;FOLD ARCON WDAT1 LIN P3 Vel=0.5 m/s CPDAT1 Tool[1]:cmttorch Base[1]:vrashatel ;%{PE}
  ;FOLD Parameters ;%{h}
    ;Params IlfProvider=kukaroboter.arctech.arconlin; Kuka.IsGlobalPoint=False; Kuka.PointName=P3; Kuka.BlendingEnabled=False; Kuka.MoveDataName=CPDAT1; Kuka.VelocityPath=0.5; Kuka.CurrentCDSetIndex=0; Kuka.MovementParameterFieldEnabled=True; ArcTech.WdatVarName=WDAT1; ArcTech.Basic=3.4.3.1264
  ;ENDFOLD
  $BWDSTART = FALSE
  LDAT_ACT = LCPDAT1
  FDAT_ACT = FP3
  BAS(#CP_PARAMS, 0.5)
  SET_CD_PARAMS (0)
  TRIGGER WHEN DISTANCE = 1 DELAY = ArcGetDelay(#PreDefinition, WDAT1) DO ArcMainNG(#PreDefinition, WDAT1, WP3) PRIO = -1
  TRIGGER WHEN PATH = ArcGetPath(#OnTheFlyArcOn, WDAT1) DELAY = ArcGetDelay(#GasPreflow, WDAT1) DO ArcMainNG(#GasPreflow, WDAT1, WP3) PRIO = -1
  TRIGGER WHEN PATH = ArcGetPath(#OnTheFlyArcOn, WDAT1) DELAY = 0 DO ArcMainNG(#ArcOnMoveStd, WDAT1, WP3) PRIO = -1
  ArcMainNG(#ArcOnBeforeMoveStd, WDAT1, WP3)
  LIN XP3
  ArcMainNG(#ArcOnAfterMoveStd, WDAT1, WP3)
;ENDFOLD
   $VEL.CP = 0.060
   LIN  {X -8.829, Y -2.041, Z 0.700, A 0.000, B 0.000, C 0.000} C_DIS

;FOLD ARCOFF WDAT2 LIN P4 CPDAT2 Tool[1]:cmttorch Base[1]:vrashatel ;%{PE}
  ;FOLD Parameters ;%{h}
    ;Params IlfProvider=kukaroboter.arctech.arcofflin; Kuka.IsGlobalPoint=False; Kuka.PointName=P4; Kuka.BlendingEnabled=False; Kuka.MoveDataName=CPDAT2; Kuka.VelocityPath=0.01; Kuka.CurrentCDSetIndex=0; Kuka.MovementParameterFieldEnabled=True; ArcTech.WdatVarName=WDAT2; ArcTech.Basic=3.4.3.1264
  ;ENDFOLD
  $BWDSTART = FALSE
  LDAT_ACT = LCPDAT2
  FDAT_ACT = FP4
  BAS(#CP_PARAMS, gArcBasVelDefinition)
  SET_CD_PARAMS (0)
  TRIGGER WHEN PATH = ArcGetPath(#ArcOffBefore, WDAT2) DELAY = 0 DO ArcMainNG(#ArcOffBeforeOffStd, WDAT2, WP4) PRIO = -1
  TRIGGER WHEN PATH = ArcGetPath(#OnTheFlyArcOff, WDAT2) DELAY = 0 DO ArcMainNG(#ArcOffMoveStd, WDAT2, WP4) PRIO = -1
  ArcMainNG(#ArcOffBeforeMoveStd, WDAT2, WP4)
  LIN XP4
  ArcMainNG(#ArcOffAfterMoveStd, WDAT2, WP4)
;ENDFOLD
   $VEL.CP = 0.080
   LIN  {X -8.829, Y -2.607, Z 0.700, A 0.000, B 0.000, C 0.000} C_DIS

;FOLD ARCON WDAT1 LIN P3 Vel=0.5 m/s CPDAT1 Tool[1]:cmttorch Base[1]:vrashatel ;%{PE}
  ;FOLD Parameters ;%{h}
    ;Params IlfProvider=kukaroboter.arctech.arconlin; Kuka.IsGlobalPoint=False; Kuka.PointName=P3; Kuka.BlendingEnabled=False; Kuka.MoveDataName=CPDAT1; Kuka.VelocityPath=0.5; Kuka.CurrentCDSetIndex=0; Kuka.MovementParameterFieldEnabled=True; ArcTech.WdatVarName=WDAT1; ArcTech.Basic=3.4.3.1264
  ;ENDFOLD
  $BWDSTART = FALSE
  LDAT_ACT = LCPDAT1
  FDAT_ACT = FP3
  BAS(#CP_PARAMS, 0.5)
  SET_CD_PARAMS (0)
  TRIGGER WHEN DISTANCE = 1 DELAY = ArcGetDelay(#PreDefinition, WDAT1) DO ArcMainNG(#PreDefinition, WDAT1, WP3) PRIO = -1
  TRIGGER WHEN PATH = ArcGetPath(#OnTheFlyArcOn, WDAT1) DELAY = ArcGetDelay(#GasPreflow, WDAT1) DO ArcMainNG(#GasPreflow, WDAT1, WP3) PRIO = -1
  TRIGGER WHEN PATH = ArcGetPath(#OnTheFlyArcOn, WDAT1) DELAY = 0 DO ArcMainNG(#ArcOnMoveStd, WDAT1, WP3) PRIO = -1
  ArcMainNG(#ArcOnBeforeMoveStd, WDAT1, WP3)
  LIN XP3
  ArcMainNG(#ArcOnAfterMoveStd, WDAT1, WP3)
;ENDFOLD
   $VEL.CP = 0.060
   LIN  {X 2.607, Y 8.829, Z 0.700, A 0.000, B 0.000, C 0.000} C_DIS

;FOLD ARCOFF WDAT2 LIN P4 CPDAT2 Tool[1]:cmttorch Base[1]:vrashatel ;%{PE}
  ;FOLD Parameters ;%{h}
    ;Params IlfProvider=kukaroboter.arctech.arcofflin; Kuka.IsGlobalPoint=False; Kuka.PointName=P4; Kuka.BlendingEnabled=False; Kuka.MoveDataName=CPDAT2; Kuka.VelocityPath=0.01; Kuka.CurrentCDSetIndex=0; Kuka.MovementParameterFieldEnabled=True; ArcTech.WdatVarName=WDAT2; ArcTech.Basic=3.4.3.1264
  ;ENDFOLD
  $BWDSTART = FALSE
  LDAT_ACT = LCPDAT2
  FDAT_ACT = FP4
  BAS(#CP_PARAMS, gArcBasVelDefinition)
  SET_CD_PARAMS (0)
  TRIGGER WHEN PATH = ArcGetPath(#ArcOffBefore, WDAT2) DELAY = 0 DO ArcMainNG(#ArcOffBeforeOffStd, WDAT2, WP4) PRIO = -1
  TRIGGER WHEN PATH = ArcGetPath(#OnTheFlyArcOff, WDAT2) DELAY = 0 DO ArcMainNG(#ArcOffMoveStd, WDAT2, WP4) PRIO = -1
  ArcMainNG(#ArcOffBeforeMoveStd, WDAT2, WP4)
  LIN XP4
  ArcMainNG(#ArcOffAfterMoveStd, WDAT2, WP4)
;ENDFOLD
   $VEL.CP = 0.080
   LIN  {X 3.172, Y 8.829, Z 0.700, A 0.000, B 0.000, C 0.000} C_DIS

;FOLD ARCON WDAT1 LIN P3 Vel=0.5 m/s CPDAT1 Tool[1]:cmttorch Base[1]:vrashatel ;%{PE}
  ;FOLD Parameters ;%{h}
    ;Params IlfProvider=kukaroboter.arctech.arconlin; Kuka.IsGlobalPoint=False; Kuka.PointName=P3; Kuka.BlendingEnabled=False; Kuka.MoveDataName=CPDAT1; Kuka.VelocityPath=0.5; Kuka.CurrentCDSetIndex=0; Kuka.MovementParameterFieldEnabled=True; ArcTech.WdatVarName=WDAT1; ArcTech.Basic=3.4.3.1264
  ;ENDFOLD
  $BWDSTART = FALSE
  LDAT_ACT = LCPDAT1
  FDAT_ACT = FP3
  BAS(#CP_PARAMS, 0.5)
  SET_CD_PARAMS (0)
  TRIGGER WHEN DISTANCE = 1 DELAY = ArcGetDelay(#PreDefinition, WDAT1) DO ArcMainNG(#PreDefinition, WDAT1, WP3) PRIO = -1
  TRIGGER WHEN PATH = ArcGetPath(#OnTheFlyArcOn, WDAT1) DELAY = ArcGetDelay(#GasPreflow, WDAT1) DO ArcMainNG(#GasPreflow, WDAT1, WP3) PRIO = -1
  TRIGGER WHEN PATH = ArcGetPath(#OnTheFlyArcOn, WDAT1) DELAY = 0 DO ArcMainNG(#ArcOnMoveStd, WDAT1, WP3) PRIO = -1
  ArcMainNG(#ArcOnBeforeMoveStd, WDAT1, WP3)
  LIN XP3
  ArcMainNG(#ArcOnAfterMoveStd, WDAT1, WP3)
;ENDFOLD
   $VEL.CP = 0.060
   LIN  {X -8.829, Y -3.172, Z 0.700, A 0.000, B 0.000, C 0.000} C_DIS

;FOLD ARCOFF WDAT2 LIN P4 CPDAT2 Tool[1]:cmttorch Base[1]:vrashatel ;%{PE}
  ;FOLD Parameters ;%{h}
    ;Params IlfProvider=kukaroboter.arctech.arcofflin; Kuka.IsGlobalPoint=False; Kuka.PointName=P4; Kuka.BlendingEnabled=False; Kuka.MoveDataName=CPDAT2; Kuka.VelocityPath=0.01; Kuka.CurrentCDSetIndex=0; Kuka.MovementParameterFieldEnabled=True; ArcTech.WdatVarName=WDAT2; ArcTech.Basic=3.4.3.1264
  ;ENDFOLD
  $BWDSTART = FALSE
  LDAT_ACT = LCPDAT2
  FDAT_ACT = FP4
  BAS(#CP_PARAMS, gArcBasVelDefinition)
  SET_CD_PARAMS (0)
  TRIGGER WHEN PATH = ArcGetPath(#ArcOffBefore, WDAT2) DELAY = 0 DO ArcMainNG(#ArcOffBeforeOffStd, WDAT2, WP4) PRIO = -1
  TRIGGER WHEN PATH = ArcGetPath(#OnTheFlyArcOff, WDAT2) DELAY = 0 DO ArcMainNG(#ArcOffMoveStd, WDAT2, WP4) PRIO = -1
  ArcMainNG(#ArcOffBeforeMoveStd, WDAT2, WP4)
  LIN XP4
  ArcMainNG(#ArcOffAfterMoveStd, WDAT2, WP4)
;ENDFOLD
   $VEL.CP = 0.080
   LIN  {X -8.829, Y -3.738, Z 0.700, A 0.000, B 0.000, C 0.000} C_DIS

;FOLD ARCON WDAT1 LIN P3 Vel=0.5 m/s CPDAT1 Tool[1]:cmttorch Base[1]:vrashatel ;%{PE}
  ;FOLD Parameters ;%{h}
    ;Params IlfProvider=kukaroboter.arctech.arconlin; Kuka.IsGlobalPoint=False; Kuka.PointName=P3; Kuka.BlendingEnabled=False; Kuka.MoveDataName=CPDAT1; Kuka.VelocityPath=0.5; Kuka.CurrentCDSetIndex=0; Kuka.MovementParameterFieldEnabled=True; ArcTech.WdatVarName=WDAT1; ArcTech.Basic=3.4.3.1264
  ;ENDFOLD
  $BWDSTART = FALSE
  LDAT_ACT = LCPDAT1
  FDAT_ACT = FP3
  BAS(#CP_PARAMS, 0.5)
  SET_CD_PARAMS (0)
  TRIGGER WHEN DISTANCE = 1 DELAY = ArcGetDelay(#PreDefinition, WDAT1) DO ArcMainNG(#PreDefinition, WDAT1, WP3) PRIO = -1
  TRIGGER WHEN PATH = ArcGetPath(#OnTheFlyArcOn, WDAT1) DELAY = ArcGetDelay(#GasPreflow, WDAT1) DO ArcMainNG(#GasPreflow, WDAT1, WP3) PRIO = -1
  TRIGGER WHEN PATH = ArcGetPath(#OnTheFlyArcOn, WDAT1) DELAY = 0 DO ArcMainNG(#ArcOnMoveStd, WDAT1, WP3) PRIO = -1
  ArcMainNG(#ArcOnBeforeMoveStd, WDAT1, WP3)
  LIN XP3
  ArcMainNG(#ArcOnAfterMoveStd, WDAT1, WP3)
;ENDFOLD
   $VEL.CP = 0.060
   LIN  {X 3.738, Y 8.829, Z 0.700, A 0.000, B 0.000, C 0.000} C_DIS

;FOLD ARCOFF WDAT2 LIN P4 CPDAT2 Tool[1]:cmttorch Base[1]:vrashatel ;%{PE}
  ;FOLD Parameters ;%{h}
    ;Params IlfProvider=kukaroboter.arctech.arcofflin; Kuka.IsGlobalPoint=False; Kuka.PointName=P4; Kuka.BlendingEnabled=False; Kuka.MoveDataName=CPDAT2; Kuka.VelocityPath=0.01; Kuka.CurrentCDSetIndex=0; Kuka.MovementParameterFieldEnabled=True; ArcTech.WdatVarName=WDAT2; ArcTech.Basic=3.4.3.1264
  ;ENDFOLD
  $BWDSTART = FALSE
  LDAT_ACT = LCPDAT2
  FDAT_ACT = FP4
  BAS(#CP_PARAMS, gArcBasVelDefinition)
  SET_CD_PARAMS (0)
  TRIGGER WHEN PATH = ArcGetPath(#ArcOffBefore, WDAT2) DELAY = 0 DO ArcMainNG(#ArcOffBeforeOffStd, WDAT2, WP4) PRIO = -1
  TRIGGER WHEN PATH = ArcGetPath(#OnTheFlyArcOff, WDAT2) DELAY = 0 DO ArcMainNG(#ArcOffMoveStd, WDAT2, WP4) PRIO = -1
  ArcMainNG(#ArcOffBeforeMoveStd, WDAT2, WP4)
  LIN XP4
  ArcMainNG(#ArcOffAfterMoveStd, WDAT2, WP4)
;ENDFOLD
   $VEL.CP = 0.080
   LIN  {X 4.304, Y 8.829, Z 0.700, A 0.000, B 0.000, C 0.000} C_DIS

;FOLD ARCON WDAT1 LIN P3 Vel=0.5 m/s CPDAT1 Tool[1]:cmttorch Base[1]:vrashatel ;%{PE}
  ;FOLD Parameters ;%{h}
    ;Params IlfProvider=kukaroboter.arctech.arconlin; Kuka.IsGlobalPoint=False; Kuka.PointName=P3; Kuka.BlendingEnabled=False; Kuka.MoveDataName=CPDAT1; Kuka.VelocityPath=0.5; Kuka.CurrentCDSetIndex=0; Kuka.MovementParameterFieldEnabled=True; ArcTech.WdatVarName=WDAT1; ArcTech.Basic=3.4.3.1264
  ;ENDFOLD
  $BWDSTART = FALSE
  LDAT_ACT = LCPDAT1
  FDAT_ACT = FP3
  BAS(#CP_PARAMS, 0.5)
  SET_CD_PARAMS (0)
  TRIGGER WHEN DISTANCE = 1 DELAY = ArcGetDelay(#PreDefinition, WDAT1) DO ArcMainNG(#PreDefinition, WDAT1, WP3) PRIO = -1
  TRIGGER WHEN PATH = ArcGetPath(#OnTheFlyArcOn, WDAT1) DELAY = ArcGetDelay(#GasPreflow, WDAT1) DO ArcMainNG(#GasPreflow, WDAT1, WP3) PRIO = -1
  TRIGGER WHEN PATH = ArcGetPath(#OnTheFlyArcOn, WDAT1) DELAY = 0 DO ArcMainNG(#ArcOnMoveStd, WDAT1, WP3) PRIO = -1
  ArcMainNG(#ArcOnBeforeMoveStd, WDAT1, WP3)
  LIN XP3
  ArcMainNG(#ArcOnAfterMoveStd, WDAT1, WP3)
;ENDFOLD
   $VEL.CP = 0.060
   LIN  {X -8.829, Y -4.304, Z 0.700, A 0.000, B 0.000, C 0.000} C_DIS

;FOLD ARCOFF WDAT2 LIN P4 CPDAT2 Tool[1]:cmttorch Base[1]:vrashatel ;%{PE}
  ;FOLD Parameters ;%{h}
    ;Params IlfProvider=kukaroboter.arctech.arcofflin; Kuka.IsGlobalPoint=False; Kuka.PointName=P4; Kuka.BlendingEnabled=False; Kuka.MoveDataName=CPDAT2; Kuka.VelocityPath=0.01; Kuka.CurrentCDSetIndex=0; Kuka.MovementParameterFieldEnabled=True; ArcTech.WdatVarName=WDAT2; ArcTech.Basic=3.4.3.1264
  ;ENDFOLD
  $BWDSTART = FALSE
  LDAT_ACT = LCPDAT2
  FDAT_ACT = FP4
  BAS(#CP_PARAMS, gArcBasVelDefinition)
  SET_CD_PARAMS (0)
  TRIGGER WHEN PATH = ArcGetPath(#ArcOffBefore, WDAT2) DELAY = 0 DO ArcMainNG(#ArcOffBeforeOffStd, WDAT2, WP4) PRIO = -1
  TRIGGER WHEN PATH = ArcGetPath(#OnTheFlyArcOff, WDAT2) DELAY = 0 DO ArcMainNG(#ArcOffMoveStd, WDAT2, WP4) PRIO = -1
  ArcMainNG(#ArcOffBeforeMoveStd, WDAT2, WP4)
  LIN XP4
  ArcMainNG(#ArcOffAfterMoveStd, WDAT2, WP4)
;ENDFOLD
   $VEL.CP = 0.080
   LIN  {X -8.829, Y -4.869, Z 0.700, A 0.000, B 0.000, C 0.000} C_DIS

;FOLD ARCON WDAT1 LIN P3 Vel=0.5 m/s CPDAT1 Tool[1]:cmttorch Base[1]:vrashatel ;%{PE}
  ;FOLD Parameters ;%{h}
    ;Params IlfProvider=kukaroboter.arctech.arconlin; Kuka.IsGlobalPoint=False; Kuka.PointName=P3; Kuka.BlendingEnabled=False; Kuka.MoveDataName=CPDAT1; Kuka.VelocityPath=0.5; Kuka.CurrentCDSetIndex=0; Kuka.MovementParameterFieldEnabled=True; ArcTech.WdatVarName=WDAT1; ArcTech.Basic=3.4.3.1264
  ;ENDFOLD
  $BWDSTART = FALSE
  LDAT_ACT = LCPDAT1
  FDAT_ACT = FP3
  BAS(#CP_PARAMS, 0.5)
  SET_CD_PARAMS (0)
  TRIGGER WHEN DISTANCE = 1 DELAY = ArcGetDelay(#PreDefinition, WDAT1) DO ArcMainNG(#PreDefinition, WDAT1, WP3) PRIO = -1
  TRIGGER WHEN PATH = ArcGetPath(#OnTheFlyArcOn, WDAT1) DELAY = ArcGetDelay(#GasPreflow, WDAT1) DO ArcMainNG(#GasPreflow, WDAT1, WP3) PRIO = -1
  TRIGGER WHEN PATH = ArcGetPath(#OnTheFlyArcOn, WDAT1) DELAY = 0 DO ArcMainNG(#ArcOnMoveStd, WDAT1, WP3) PRIO = -1
  ArcMainNG(#ArcOnBeforeMoveStd, WDAT1, WP3)
  LIN XP3
  ArcMainNG(#ArcOnAfterMoveStd, WDAT1, WP3)
;ENDFOLD
   $VEL.CP = 0.060
   LIN  {X 4.869, Y 8.829, Z 0.700, A 0.000, B 0.000, C 0.000} C_DIS

;FOLD ARCOFF WDAT2 LIN P4 CPDAT2 Tool[1]:cmttorch Base[1]:vrashatel ;%{PE}
  ;FOLD Parameters ;%{h}
    ;Params IlfProvider=kukaroboter.arctech.arcofflin; Kuka.IsGlobalPoint=False; Kuka.PointName=P4; Kuka.BlendingEnabled=False; Kuka.MoveDataName=CPDAT2; Kuka.VelocityPath=0.01; Kuka.CurrentCDSetIndex=0; Kuka.MovementParameterFieldEnabled=True; ArcTech.WdatVarName=WDAT2; ArcTech.Basic=3.4.3.1264
  ;ENDFOLD
  $BWDSTART = FALSE
  LDAT_ACT = LCPDAT2
  FDAT_ACT = FP4
  BAS(#CP_PARAMS, gArcBasVelDefinition)
  SET_CD_PARAMS (0)
  TRIGGER WHEN PATH = ArcGetPath(#ArcOffBefore, WDAT2) DELAY = 0 DO ArcMainNG(#ArcOffBeforeOffStd, WDAT2, WP4) PRIO = -1
  TRIGGER WHEN PATH = ArcGetPath(#OnTheFlyArcOff, WDAT2) DELAY = 0 DO ArcMainNG(#ArcOffMoveStd, WDAT2, WP4) PRIO = -1
  ArcMainNG(#ArcOffBeforeMoveStd, WDAT2, WP4)
  LIN XP4
  ArcMainNG(#ArcOffAfterMoveStd, WDAT2, WP4)
;ENDFOLD
   $VEL.CP = 0.080
   LIN  {X 5.435, Y 8.829, Z 0.700, A 0.000, B 0.000, C 0.000} C_DIS

;FOLD ARCON WDAT1 LIN P3 Vel=0.5 m/s CPDAT1 Tool[1]:cmttorch Base[1]:vrashatel ;%{PE}
  ;FOLD Parameters ;%{h}
    ;Params IlfProvider=kukaroboter.arctech.arconlin; Kuka.IsGlobalPoint=False; Kuka.PointName=P3; Kuka.BlendingEnabled=False; Kuka.MoveDataName=CPDAT1; Kuka.VelocityPath=0.5; Kuka.CurrentCDSetIndex=0; Kuka.MovementParameterFieldEnabled=True; ArcTech.WdatVarName=WDAT1; ArcTech.Basic=3.4.3.1264
  ;ENDFOLD
  $BWDSTART = FALSE
  LDAT_ACT = LCPDAT1
  FDAT_ACT = FP3
  BAS(#CP_PARAMS, 0.5)
  SET_CD_PARAMS (0)
  TRIGGER WHEN DISTANCE = 1 DELAY = ArcGetDelay(#PreDefinition, WDAT1) DO ArcMainNG(#PreDefinition, WDAT1, WP3) PRIO = -1
  TRIGGER WHEN PATH = ArcGetPath(#OnTheFlyArcOn, WDAT1) DELAY = ArcGetDelay(#GasPreflow, WDAT1) DO ArcMainNG(#GasPreflow, WDAT1, WP3) PRIO = -1
  TRIGGER WHEN PATH = ArcGetPath(#OnTheFlyArcOn, WDAT1) DELAY = 0 DO ArcMainNG(#ArcOnMoveStd, WDAT1, WP3) PRIO = -1
  ArcMainNG(#ArcOnBeforeMoveStd, WDAT1, WP3)
  LIN XP3
  ArcMainNG(#ArcOnAfterMoveStd, WDAT1, WP3)
;ENDFOLD
   $VEL.CP = 0.060
   LIN  {X -8.829, Y -5.435, Z 0.700, A 0.000, B 0.000, C 0.000} C_DIS

;FOLD ARCOFF WDAT2 LIN P4 CPDAT2 Tool[1]:cmttorch Base[1]:vrashatel ;%{PE}
  ;FOLD Parameters ;%{h}
    ;Params IlfProvider=kukaroboter.arctech.arcofflin; Kuka.IsGlobalPoint=False; Kuka.PointName=P4; Kuka.BlendingEnabled=False; Kuka.MoveDataName=CPDAT2; Kuka.VelocityPath=0.01; Kuka.CurrentCDSetIndex=0; Kuka.MovementParameterFieldEnabled=True; ArcTech.WdatVarName=WDAT2; ArcTech.Basic=3.4.3.1264
  ;ENDFOLD
  $BWDSTART = FALSE
  LDAT_ACT = LCPDAT2
  FDAT_ACT = FP4
  BAS(#CP_PARAMS, gArcBasVelDefinition)
  SET_CD_PARAMS (0)
  TRIGGER WHEN PATH = ArcGetPath(#ArcOffBefore, WDAT2) DELAY = 0 DO ArcMainNG(#ArcOffBeforeOffStd, WDAT2, WP4) PRIO = -1
  TRIGGER WHEN PATH = ArcGetPath(#OnTheFlyArcOff, WDAT2) DELAY = 0 DO ArcMainNG(#ArcOffMoveStd, WDAT2, WP4) PRIO = -1
  ArcMainNG(#ArcOffBeforeMoveStd, WDAT2, WP4)
  LIN XP4
  ArcMainNG(#ArcOffAfterMoveStd, WDAT2, WP4)
;ENDFOLD
   $VEL.CP = 0.080
   LIN  {X -8.829, Y -6.001, Z 0.700, A 0.000, B 0.000, C 0.000} C_DIS

;FOLD ARCON WDAT1 LIN P3 Vel=0.5 m/s CPDAT1 Tool[1]:cmttorch Base[1]:vrashatel ;%{PE}
  ;FOLD Parameters ;%{h}
    ;Params IlfProvider=kukaroboter.arctech.arconlin; Kuka.IsGlobalPoint=False; Kuka.PointName=P3; Kuka.BlendingEnabled=False; Kuka.MoveDataName=CPDAT1; Kuka.VelocityPath=0.5; Kuka.CurrentCDSetIndex=0; Kuka.MovementParameterFieldEnabled=True; ArcTech.WdatVarName=WDAT1; ArcTech.Basic=3.4.3.1264
  ;ENDFOLD
  $BWDSTART = FALSE
  LDAT_ACT = LCPDAT1
  FDAT_ACT = FP3
  BAS(#CP_PARAMS, 0.5)
  SET_CD_PARAMS (0)
  TRIGGER WHEN DISTANCE = 1 DELAY = ArcGetDelay(#PreDefinition, WDAT1) DO ArcMainNG(#PreDefinition, WDAT1, WP3) PRIO = -1
  TRIGGER WHEN PATH = ArcGetPath(#OnTheFlyArcOn, WDAT1) DELAY = ArcGetDelay(#GasPreflow, WDAT1) DO ArcMainNG(#GasPreflow, WDAT1, WP3) PRIO = -1
  TRIGGER WHEN PATH = ArcGetPath(#OnTheFlyArcOn, WDAT1) DELAY = 0 DO ArcMainNG(#ArcOnMoveStd, WDAT1, WP3) PRIO = -1
  ArcMainNG(#ArcOnBeforeMoveStd, WDAT1, WP3)
  LIN XP3
  ArcMainNG(#ArcOnAfterMoveStd, WDAT1, WP3)
;ENDFOLD
   $VEL.CP = 0.060
   LIN  {X 6.001, Y 8.829, Z 0.700, A 0.000, B 0.000, C 0.000} C_DIS

;FOLD ARCOFF WDAT2 LIN P4 CPDAT2 Tool[1]:cmttorch Base[1]:vrashatel ;%{PE}
  ;FOLD Parameters ;%{h}
    ;Params IlfProvider=kukaroboter.arctech.arcofflin; Kuka.IsGlobalPoint=False; Kuka.PointName=P4; Kuka.BlendingEnabled=False; Kuka.MoveDataName=CPDAT2; Kuka.VelocityPath=0.01; Kuka.CurrentCDSetIndex=0; Kuka.MovementParameterFieldEnabled=True; ArcTech.WdatVarName=WDAT2; ArcTech.Basic=3.4.3.1264
  ;ENDFOLD
  $BWDSTART = FALSE
  LDAT_ACT = LCPDAT2
  FDAT_ACT = FP4
  BAS(#CP_PARAMS, gArcBasVelDefinition)
  SET_CD_PARAMS (0)
  TRIGGER WHEN PATH = ArcGetPath(#ArcOffBefore, WDAT2) DELAY = 0 DO ArcMainNG(#ArcOffBeforeOffStd, WDAT2, WP4) PRIO = -1
  TRIGGER WHEN PATH = ArcGetPath(#OnTheFlyArcOff, WDAT2) DELAY = 0 DO ArcMainNG(#ArcOffMoveStd, WDAT2, WP4) PRIO = -1
  ArcMainNG(#ArcOffBeforeMoveStd, WDAT2, WP4)
  LIN XP4
  ArcMainNG(#ArcOffAfterMoveStd, WDAT2, WP4)
;ENDFOLD
   $VEL.CP = 0.080
   LIN  {X 6.566, Y 8.829, Z 0.700, A 0.000, B 0.000, C 0.000} C_DIS

;FOLD ARCON WDAT1 LIN P3 Vel=0.5 m/s CPDAT1 Tool[1]:cmttorch Base[1]:vrashatel ;%{PE}
  ;FOLD Parameters ;%{h}
    ;Params IlfProvider=kukaroboter.arctech.arconlin; Kuka.IsGlobalPoint=False; Kuka.PointName=P3; Kuka.BlendingEnabled=False; Kuka.MoveDataName=CPDAT1; Kuka.VelocityPath=0.5; Kuka.CurrentCDSetIndex=0; Kuka.MovementParameterFieldEnabled=True; ArcTech.WdatVarName=WDAT1; ArcTech.Basic=3.4.3.1264
  ;ENDFOLD
  $BWDSTART = FALSE
  LDAT_ACT = LCPDAT1
  FDAT_ACT = FP3
  BAS(#CP_PARAMS, 0.5)
  SET_CD_PARAMS (0)
  TRIGGER WHEN DISTANCE = 1 DELAY = ArcGetDelay(#PreDefinition, WDAT1) DO ArcMainNG(#PreDefinition, WDAT1, WP3) PRIO = -1
  TRIGGER WHEN PATH = ArcGetPath(#OnTheFlyArcOn, WDAT1) DELAY = ArcGetDelay(#GasPreflow, WDAT1) DO ArcMainNG(#GasPreflow, WDAT1, WP3) PRIO = -1
  TRIGGER WHEN PATH = ArcGetPath(#OnTheFlyArcOn, WDAT1) DELAY = 0 DO ArcMainNG(#ArcOnMoveStd, WDAT1, WP3) PRIO = -1
  ArcMainNG(#ArcOnBeforeMoveStd, WDAT1, WP3)
  LIN XP3
  ArcMainNG(#ArcOnAfterMoveStd, WDAT1, WP3)
;ENDFOLD
   $VEL.CP = 0.060
   LIN  {X -8.829, Y -6.566, Z 0.700, A 0.000, B 0.000, C 0.000} C_DIS

;FOLD ARCOFF WDAT2 LIN P4 CPDAT2 Tool[1]:cmttorch Base[1]:vrashatel ;%{PE}
  ;FOLD Parameters ;%{h}
    ;Params IlfProvider=kukaroboter.arctech.arcofflin; Kuka.IsGlobalPoint=False; Kuka.PointName=P4; Kuka.BlendingEnabled=False; Kuka.MoveDataName=CPDAT2; Kuka.VelocityPath=0.01; Kuka.CurrentCDSetIndex=0; Kuka.MovementParameterFieldEnabled=True; ArcTech.WdatVarName=WDAT2; ArcTech.Basic=3.4.3.1264
  ;ENDFOLD
  $BWDSTART = FALSE
  LDAT_ACT = LCPDAT2
  FDAT_ACT = FP4
  BAS(#CP_PARAMS, gArcBasVelDefinition)
  SET_CD_PARAMS (0)
  TRIGGER WHEN PATH = ArcGetPath(#ArcOffBefore, WDAT2) DELAY = 0 DO ArcMainNG(#ArcOffBeforeOffStd, WDAT2, WP4) PRIO = -1
  TRIGGER WHEN PATH = ArcGetPath(#OnTheFlyArcOff, WDAT2) DELAY = 0 DO ArcMainNG(#ArcOffMoveStd, WDAT2, WP4) PRIO = -1
  ArcMainNG(#ArcOffBeforeMoveStd, WDAT2, WP4)
  LIN XP4
  ArcMainNG(#ArcOffAfterMoveStd, WDAT2, WP4)
;ENDFOLD
   $VEL.CP = 0.080
   LIN  {X -8.829, Y -7.132, Z 0.700, A 0.000, B 0.000, C 0.000} C_DIS

;FOLD ARCON WDAT1 LIN P3 Vel=0.5 m/s CPDAT1 Tool[1]:cmttorch Base[1]:vrashatel ;%{PE}
  ;FOLD Parameters ;%{h}
    ;Params IlfProvider=kukaroboter.arctech.arconlin; Kuka.IsGlobalPoint=False; Kuka.PointName=P3; Kuka.BlendingEnabled=False; Kuka.MoveDataName=CPDAT1; Kuka.VelocityPath=0.5; Kuka.CurrentCDSetIndex=0; Kuka.MovementParameterFieldEnabled=True; ArcTech.WdatVarName=WDAT1; ArcTech.Basic=3.4.3.1264
  ;ENDFOLD
  $BWDSTART = FALSE
  LDAT_ACT = LCPDAT1
  FDAT_ACT = FP3
  BAS(#CP_PARAMS, 0.5)
  SET_CD_PARAMS (0)
  TRIGGER WHEN DISTANCE = 1 DELAY = ArcGetDelay(#PreDefinition, WDAT1) DO ArcMainNG(#PreDefinition, WDAT1, WP3) PRIO = -1
  TRIGGER WHEN PATH = ArcGetPath(#OnTheFlyArcOn, WDAT1) DELAY = ArcGetDelay(#GasPreflow, WDAT1) DO ArcMainNG(#GasPreflow, WDAT1, WP3) PRIO = -1
  TRIGGER WHEN PATH = ArcGetPath(#OnTheFlyArcOn, WDAT1) DELAY = 0 DO ArcMainNG(#ArcOnMoveStd, WDAT1, WP3) PRIO = -1
  ArcMainNG(#ArcOnBeforeMoveStd, WDAT1, WP3)
  LIN XP3
  ArcMainNG(#ArcOnAfterMoveStd, WDAT1, WP3)
;ENDFOLD
   $VEL.CP = 0.060
   LIN  {X 7.132, Y 8.829, Z 0.700, A 0.000, B 0.000, C 0.000} C_DIS

;FOLD ARCOFF WDAT2 LIN P4 CPDAT2 Tool[1]:cmttorch Base[1]:vrashatel ;%{PE}
  ;FOLD Parameters ;%{h}
    ;Params IlfProvider=kukaroboter.arctech.arcofflin; Kuka.IsGlobalPoint=False; Kuka.PointName=P4; Kuka.BlendingEnabled=False; Kuka.MoveDataName=CPDAT2; Kuka.VelocityPath=0.01; Kuka.CurrentCDSetIndex=0; Kuka.MovementParameterFieldEnabled=True; ArcTech.WdatVarName=WDAT2; ArcTech.Basic=3.4.3.1264
  ;ENDFOLD
  $BWDSTART = FALSE
  LDAT_ACT = LCPDAT2
  FDAT_ACT = FP4
  BAS(#CP_PARAMS, gArcBasVelDefinition)
  SET_CD_PARAMS (0)
  TRIGGER WHEN PATH = ArcGetPath(#ArcOffBefore, WDAT2) DELAY = 0 DO ArcMainNG(#ArcOffBeforeOffStd, WDAT2, WP4) PRIO = -1
  TRIGGER WHEN PATH = ArcGetPath(#OnTheFlyArcOff, WDAT2) DELAY = 0 DO ArcMainNG(#ArcOffMoveStd, WDAT2, WP4) PRIO = -1
  ArcMainNG(#ArcOffBeforeMoveStd, WDAT2, WP4)
  LIN XP4
  ArcMainNG(#ArcOffAfterMoveStd, WDAT2, WP4)
;ENDFOLD
   $VEL.CP = 0.080
   LIN  {X 7.698, Y 8.829, Z 0.700, A 0.000, B 0.000, C 0.000} C_DIS

;FOLD ARCON WDAT1 LIN P3 Vel=0.5 m/s CPDAT1 Tool[1]:cmttorch Base[1]:vrashatel ;%{PE}
  ;FOLD Parameters ;%{h}
    ;Params IlfProvider=kukaroboter.arctech.arconlin; Kuka.IsGlobalPoint=False; Kuka.PointName=P3; Kuka.BlendingEnabled=False; Kuka.MoveDataName=CPDAT1; Kuka.VelocityPath=0.5; Kuka.CurrentCDSetIndex=0; Kuka.MovementParameterFieldEnabled=True; ArcTech.WdatVarName=WDAT1; ArcTech.Basic=3.4.3.1264
  ;ENDFOLD
  $BWDSTART = FALSE
  LDAT_ACT = LCPDAT1
  FDAT_ACT = FP3
  BAS(#CP_PARAMS, 0.5)
  SET_CD_PARAMS (0)
  TRIGGER WHEN DISTANCE = 1 DELAY = ArcGetDelay(#PreDefinition, WDAT1) DO ArcMainNG(#PreDefinition, WDAT1, WP3) PRIO = -1
  TRIGGER WHEN PATH = ArcGetPath(#OnTheFlyArcOn, WDAT1) DELAY = ArcGetDelay(#GasPreflow, WDAT1) DO ArcMainNG(#GasPreflow, WDAT1, WP3) PRIO = -1
  TRIGGER WHEN PATH = ArcGetPath(#OnTheFlyArcOn, WDAT1) DELAY = 0 DO ArcMainNG(#ArcOnMoveStd, WDAT1, WP3) PRIO = -1
  ArcMainNG(#ArcOnBeforeMoveStd, WDAT1, WP3)
  LIN XP3
  ArcMainNG(#ArcOnAfterMoveStd, WDAT1, WP3)
;ENDFOLD
   $VEL.CP = 0.060
   LIN  {X -8.829, Y -7.698, Z 0.700, A 0.000, B 0.000, C 0.000} C_DIS

;FOLD ARCOFF WDAT2 LIN P4 CPDAT2 Tool[1]:cmttorch Base[1]:vrashatel ;%{PE}
  ;FOLD Parameters ;%{h}
    ;Params IlfProvider=kukaroboter.arctech.arcofflin; Kuka.IsGlobalPoint=False; Kuka.PointName=P4; Kuka.BlendingEnabled=False; Kuka.MoveDataName=CPDAT2; Kuka.VelocityPath=0.01; Kuka.CurrentCDSetIndex=0; Kuka.MovementParameterFieldEnabled=True; ArcTech.WdatVarName=WDAT2; ArcTech.Basic=3.4.3.1264
  ;ENDFOLD
  $BWDSTART = FALSE
  LDAT_ACT = LCPDAT2
  FDAT_ACT = FP4
  BAS(#CP_PARAMS, gArcBasVelDefinition)
  SET_CD_PARAMS (0)
  TRIGGER WHEN PATH = ArcGetPath(#ArcOffBefore, WDAT2) DELAY = 0 DO ArcMainNG(#ArcOffBeforeOffStd, WDAT2, WP4) PRIO = -1
  TRIGGER WHEN PATH = ArcGetPath(#OnTheFlyArcOff, WDAT2) DELAY = 0 DO ArcMainNG(#ArcOffMoveStd, WDAT2, WP4) PRIO = -1
  ArcMainNG(#ArcOffBeforeMoveStd, WDAT2, WP4)
  LIN XP4
  ArcMainNG(#ArcOffAfterMoveStd, WDAT2, WP4)
;ENDFOLD
   $VEL.CP = 0.080
   LIN  {X -8.829, Y -8.263, Z 0.700, A 0.000, B 0.000, C 0.000} C_DIS

;FOLD ARCON WDAT1 LIN P3 Vel=0.5 m/s CPDAT1 Tool[1]:cmttorch Base[1]:vrashatel ;%{PE}
  ;FOLD Parameters ;%{h}
    ;Params IlfProvider=kukaroboter.arctech.arconlin; Kuka.IsGlobalPoint=False; Kuka.PointName=P3; Kuka.BlendingEnabled=False; Kuka.MoveDataName=CPDAT1; Kuka.VelocityPath=0.5; Kuka.CurrentCDSetIndex=0; Kuka.MovementParameterFieldEnabled=True; ArcTech.WdatVarName=WDAT1; ArcTech.Basic=3.4.3.1264
  ;ENDFOLD
  $BWDSTART = FALSE
  LDAT_ACT = LCPDAT1
  FDAT_ACT = FP3
  BAS(#CP_PARAMS, 0.5)
  SET_CD_PARAMS (0)
  TRIGGER WHEN DISTANCE = 1 DELAY = ArcGetDelay(#PreDefinition, WDAT1) DO ArcMainNG(#PreDefinition, WDAT1, WP3) PRIO = -1
  TRIGGER WHEN PATH = ArcGetPath(#OnTheFlyArcOn, WDAT1) DELAY = ArcGetDelay(#GasPreflow, WDAT1) DO ArcMainNG(#GasPreflow, WDAT1, WP3) PRIO = -1
  TRIGGER WHEN PATH = ArcGetPath(#OnTheFlyArcOn, WDAT1) DELAY = 0 DO ArcMainNG(#ArcOnMoveStd, WDAT1, WP3) PRIO = -1
  ArcMainNG(#ArcOnBeforeMoveStd, WDAT1, WP3)
  LIN XP3
  ArcMainNG(#ArcOnAfterMoveStd, WDAT1, WP3)
;ENDFOLD
   $VEL.CP = 0.060
   LIN  {X 8.263, Y 8.829, Z 0.700, A 0.000, B 0.000, C 0.000} C_DIS

;FOLD ARCOFF WDAT2 LIN P4 CPDAT2 Tool[1]:cmttorch Base[1]:vrashatel ;%{PE}
  ;FOLD Parameters ;%{h}
    ;Params IlfProvider=kukaroboter.arctech.arcofflin; Kuka.IsGlobalPoint=False; Kuka.PointName=P4; Kuka.BlendingEnabled=False; Kuka.MoveDataName=CPDAT2; Kuka.VelocityPath=0.01; Kuka.CurrentCDSetIndex=0; Kuka.MovementParameterFieldEnabled=True; ArcTech.WdatVarName=WDAT2; ArcTech.Basic=3.4.3.1264
  ;ENDFOLD
  $BWDSTART = FALSE
  LDAT_ACT = LCPDAT2
  FDAT_ACT = FP4
  BAS(#CP_PARAMS, gArcBasVelDefinition)
  SET_CD_PARAMS (0)
  TRIGGER WHEN PATH = ArcGetPath(#ArcOffBefore, WDAT2) DELAY = 0 DO ArcMainNG(#ArcOffBeforeOffStd, WDAT2, WP4) PRIO = -1
  TRIGGER WHEN PATH = ArcGetPath(#OnTheFlyArcOff, WDAT2) DELAY = 0 DO ArcMainNG(#ArcOffMoveStd, WDAT2, WP4) PRIO = -1
  ArcMainNG(#ArcOffBeforeMoveStd, WDAT2, WP4)
  LIN XP4
  ArcMainNG(#ArcOffAfterMoveStd, WDAT2, WP4)
;ENDFOLD
   $VEL.CP = 0.080
   LIN  {X 8.829, Y 8.829, Z 0.700, A 0.000, B 0.000, C 0.000} C_DIS

;FOLD ARCON WDAT1 LIN P3 Vel=0.5 m/s CPDAT1 Tool[1]:cmttorch Base[1]:vrashatel ;%{PE}
  ;FOLD Parameters ;%{h}
    ;Params IlfProvider=kukaroboter.arctech.arconlin; Kuka.IsGlobalPoint=False; Kuka.PointName=P3; Kuka.BlendingEnabled=False; Kuka.MoveDataName=CPDAT1; Kuka.VelocityPath=0.5; Kuka.CurrentCDSetIndex=0; Kuka.MovementParameterFieldEnabled=True; ArcTech.WdatVarName=WDAT1; ArcTech.Basic=3.4.3.1264
  ;ENDFOLD
  $BWDSTART = FALSE
  LDAT_ACT = LCPDAT1
  FDAT_ACT = FP3
  BAS(#CP_PARAMS, 0.5)
  SET_CD_PARAMS (0)
  TRIGGER WHEN DISTANCE = 1 DELAY = ArcGetDelay(#PreDefinition, WDAT1) DO ArcMainNG(#PreDefinition, WDAT1, WP3) PRIO = -1
  TRIGGER WHEN PATH = ArcGetPath(#OnTheFlyArcOn, WDAT1) DELAY = ArcGetDelay(#GasPreflow, WDAT1) DO ArcMainNG(#GasPreflow, WDAT1, WP3) PRIO = -1
  TRIGGER WHEN PATH = ArcGetPath(#OnTheFlyArcOn, WDAT1) DELAY = 0 DO ArcMainNG(#ArcOnMoveStd, WDAT1, WP3) PRIO = -1
  ArcMainNG(#ArcOnBeforeMoveStd, WDAT1, WP3)
  LIN XP3
  ArcMainNG(#ArcOnAfterMoveStd, WDAT1, WP3)
;ENDFOLD
   $VEL.CP = 0.060
   LIN  {X -8.829, Y -8.829, Z 0.700, A 0.000, B 0.000, C 0.000} C_DIS

;FOLD ARCOFF WDAT2 LIN P4 CPDAT2 Tool[1]:cmttorch Base[1]:vrashatel ;%{PE}
  ;FOLD Parameters ;%{h}
    ;Params IlfProvider=kukaroboter.arctech.arcofflin; Kuka.IsGlobalPoint=False; Kuka.PointName=P4; Kuka.BlendingEnabled=False; Kuka.MoveDataName=CPDAT2; Kuka.VelocityPath=0.01; Kuka.CurrentCDSetIndex=0; Kuka.MovementParameterFieldEnabled=True; ArcTech.WdatVarName=WDAT2; ArcTech.Basic=3.4.3.1264
  ;ENDFOLD
  $BWDSTART = FALSE
  LDAT_ACT = LCPDAT2
  FDAT_ACT = FP4
  BAS(#CP_PARAMS, gArcBasVelDefinition)
  SET_CD_PARAMS (0)
  TRIGGER WHEN PATH = ArcGetPath(#ArcOffBefore, WDAT2) DELAY = 0 DO ArcMainNG(#ArcOffBeforeOffStd, WDAT2, WP4) PRIO = -1
  TRIGGER WHEN PATH = ArcGetPath(#OnTheFlyArcOff, WDAT2) DELAY = 0 DO ArcMainNG(#ArcOffMoveStd, WDAT2, WP4) PRIO = -1
  ArcMainNG(#ArcOffBeforeMoveStd, WDAT2, WP4)
  LIN XP4
  ArcMainNG(#ArcOffAfterMoveStd, WDAT2, WP4)
;ENDFOLD
   $VEL.CP = 0.080
   LIN  {X -8.263, Y -8.829, Z 0.700, A 0.000, B 0.000, C 0.000} C_DIS

;FOLD ARCON WDAT1 LIN P3 Vel=0.5 m/s CPDAT1 Tool[1]:cmttorch Base[1]:vrashatel ;%{PE}
  ;FOLD Parameters ;%{h}
    ;Params IlfProvider=kukaroboter.arctech.arconlin; Kuka.IsGlobalPoint=False; Kuka.PointName=P3; Kuka.BlendingEnabled=False; Kuka.MoveDataName=CPDAT1; Kuka.VelocityPath=0.5; Kuka.CurrentCDSetIndex=0; Kuka.MovementParameterFieldEnabled=True; ArcTech.WdatVarName=WDAT1; ArcTech.Basic=3.4.3.1264
  ;ENDFOLD
  $BWDSTART = FALSE
  LDAT_ACT = LCPDAT1
  FDAT_ACT = FP3
  BAS(#CP_PARAMS, 0.5)
  SET_CD_PARAMS (0)
  TRIGGER WHEN DISTANCE = 1 DELAY = ArcGetDelay(#PreDefinition, WDAT1) DO ArcMainNG(#PreDefinition, WDAT1, WP3) PRIO = -1
  TRIGGER WHEN PATH = ArcGetPath(#OnTheFlyArcOn, WDAT1) DELAY = ArcGetDelay(#GasPreflow, WDAT1) DO ArcMainNG(#GasPreflow, WDAT1, WP3) PRIO = -1
  TRIGGER WHEN PATH = ArcGetPath(#OnTheFlyArcOn, WDAT1) DELAY = 0 DO ArcMainNG(#ArcOnMoveStd, WDAT1, WP3) PRIO = -1
  ArcMainNG(#ArcOnBeforeMoveStd, WDAT1, WP3)
  LIN XP3
  ArcMainNG(#ArcOnAfterMoveStd, WDAT1, WP3)
;ENDFOLD
   $VEL.CP = 0.060
   LIN  {X 8.829, Y 8.263, Z 0.700, A 0.000, B 0.000, C 0.000} C_DIS

;FOLD ARCOFF WDAT2 LIN P4 CPDAT2 Tool[1]:cmttorch Base[1]:vrashatel ;%{PE}
  ;FOLD Parameters ;%{h}
    ;Params IlfProvider=kukaroboter.arctech.arcofflin; Kuka.IsGlobalPoint=False; Kuka.PointName=P4; Kuka.BlendingEnabled=False; Kuka.MoveDataName=CPDAT2; Kuka.VelocityPath=0.01; Kuka.CurrentCDSetIndex=0; Kuka.MovementParameterFieldEnabled=True; ArcTech.WdatVarName=WDAT2; ArcTech.Basic=3.4.3.1264
  ;ENDFOLD
  $BWDSTART = FALSE
  LDAT_ACT = LCPDAT2
  FDAT_ACT = FP4
  BAS(#CP_PARAMS, gArcBasVelDefinition)
  SET_CD_PARAMS (0)
  TRIGGER WHEN PATH = ArcGetPath(#ArcOffBefore, WDAT2) DELAY = 0 DO ArcMainNG(#ArcOffBeforeOffStd, WDAT2, WP4) PRIO = -1
  TRIGGER WHEN PATH = ArcGetPath(#OnTheFlyArcOff, WDAT2) DELAY = 0 DO ArcMainNG(#ArcOffMoveStd, WDAT2, WP4) PRIO = -1
  ArcMainNG(#ArcOffBeforeMoveStd, WDAT2, WP4)
  LIN XP4
  ArcMainNG(#ArcOffAfterMoveStd, WDAT2, WP4)
;ENDFOLD
   $VEL.CP = 0.080
   LIN  {X 8.829, Y 7.698, Z 0.700, A 0.000, B 0.000, C 0.000} C_DIS

;FOLD ARCON WDAT1 LIN P3 Vel=0.5 m/s CPDAT1 Tool[1]:cmttorch Base[1]:vrashatel ;%{PE}
  ;FOLD Parameters ;%{h}
    ;Params IlfProvider=kukaroboter.arctech.arconlin; Kuka.IsGlobalPoint=False; Kuka.PointName=P3; Kuka.BlendingEnabled=False; Kuka.MoveDataName=CPDAT1; Kuka.VelocityPath=0.5; Kuka.CurrentCDSetIndex=0; Kuka.MovementParameterFieldEnabled=True; ArcTech.WdatVarName=WDAT1; ArcTech.Basic=3.4.3.1264
  ;ENDFOLD
  $BWDSTART = FALSE
  LDAT_ACT = LCPDAT1
  FDAT_ACT = FP3
  BAS(#CP_PARAMS, 0.5)
  SET_CD_PARAMS (0)
  TRIGGER WHEN DISTANCE = 1 DELAY = ArcGetDelay(#PreDefinition, WDAT1) DO ArcMainNG(#PreDefinition, WDAT1, WP3) PRIO = -1
  TRIGGER WHEN PATH = ArcGetPath(#OnTheFlyArcOn, WDAT1) DELAY = ArcGetDelay(#GasPreflow, WDAT1) DO ArcMainNG(#GasPreflow, WDAT1, WP3) PRIO = -1
  TRIGGER WHEN PATH = ArcGetPath(#OnTheFlyArcOn, WDAT1) DELAY = 0 DO ArcMainNG(#ArcOnMoveStd, WDAT1, WP3) PRIO = -1
  ArcMainNG(#ArcOnBeforeMoveStd, WDAT1, WP3)
  LIN XP3
  ArcMainNG(#ArcOnAfterMoveStd, WDAT1, WP3)
;ENDFOLD
   $VEL.CP = 0.060
   LIN  {X -7.698, Y -8.829, Z 0.700, A 0.000, B 0.000, C 0.000} C_DIS

;FOLD ARCOFF WDAT2 LIN P4 CPDAT2 Tool[1]:cmttorch Base[1]:vrashatel ;%{PE}
  ;FOLD Parameters ;%{h}
    ;Params IlfProvider=kukaroboter.arctech.arcofflin; Kuka.IsGlobalPoint=False; Kuka.PointName=P4; Kuka.BlendingEnabled=False; Kuka.MoveDataName=CPDAT2; Kuka.VelocityPath=0.01; Kuka.CurrentCDSetIndex=0; Kuka.MovementParameterFieldEnabled=True; ArcTech.WdatVarName=WDAT2; ArcTech.Basic=3.4.3.1264
  ;ENDFOLD
  $BWDSTART = FALSE
  LDAT_ACT = LCPDAT2
  FDAT_ACT = FP4
  BAS(#CP_PARAMS, gArcBasVelDefinition)
  SET_CD_PARAMS (0)
  TRIGGER WHEN PATH = ArcGetPath(#ArcOffBefore, WDAT2) DELAY = 0 DO ArcMainNG(#ArcOffBeforeOffStd, WDAT2, WP4) PRIO = -1
  TRIGGER WHEN PATH = ArcGetPath(#OnTheFlyArcOff, WDAT2) DELAY = 0 DO ArcMainNG(#ArcOffMoveStd, WDAT2, WP4) PRIO = -1
  ArcMainNG(#ArcOffBeforeMoveStd, WDAT2, WP4)
  LIN XP4
  ArcMainNG(#ArcOffAfterMoveStd, WDAT2, WP4)
;ENDFOLD
   $VEL.CP = 0.080
   LIN  {X -7.132, Y -8.829, Z 0.700, A 0.000, B 0.000, C 0.000} C_DIS

;FOLD ARCON WDAT1 LIN P3 Vel=0.5 m/s CPDAT1 Tool[1]:cmttorch Base[1]:vrashatel ;%{PE}
  ;FOLD Parameters ;%{h}
    ;Params IlfProvider=kukaroboter.arctech.arconlin; Kuka.IsGlobalPoint=False; Kuka.PointName=P3; Kuka.BlendingEnabled=False; Kuka.MoveDataName=CPDAT1; Kuka.VelocityPath=0.5; Kuka.CurrentCDSetIndex=0; Kuka.MovementParameterFieldEnabled=True; ArcTech.WdatVarName=WDAT1; ArcTech.Basic=3.4.3.1264
  ;ENDFOLD
  $BWDSTART = FALSE
  LDAT_ACT = LCPDAT1
  FDAT_ACT = FP3
  BAS(#CP_PARAMS, 0.5)
  SET_CD_PARAMS (0)
  TRIGGER WHEN DISTANCE = 1 DELAY = ArcGetDelay(#PreDefinition, WDAT1) DO ArcMainNG(#PreDefinition, WDAT1, WP3) PRIO = -1
  TRIGGER WHEN PATH = ArcGetPath(#OnTheFlyArcOn, WDAT1) DELAY = ArcGetDelay(#GasPreflow, WDAT1) DO ArcMainNG(#GasPreflow, WDAT1, WP3) PRIO = -1
  TRIGGER WHEN PATH = ArcGetPath(#OnTheFlyArcOn, WDAT1) DELAY = 0 DO ArcMainNG(#ArcOnMoveStd, WDAT1, WP3) PRIO = -1
  ArcMainNG(#ArcOnBeforeMoveStd, WDAT1, WP3)
  LIN XP3
  ArcMainNG(#ArcOnAfterMoveStd, WDAT1, WP3)
;ENDFOLD
   $VEL.CP = 0.060
   LIN  {X 8.829, Y 7.132, Z 0.700, A 0.000, B 0.000, C 0.000} C_DIS

;FOLD ARCOFF WDAT2 LIN P4 CPDAT2 Tool[1]:cmttorch Base[1]:vrashatel ;%{PE}
  ;FOLD Parameters ;%{h}
    ;Params IlfProvider=kukaroboter.arctech.arcofflin; Kuka.IsGlobalPoint=False; Kuka.PointName=P4; Kuka.BlendingEnabled=False; Kuka.MoveDataName=CPDAT2; Kuka.VelocityPath=0.01; Kuka.CurrentCDSetIndex=0; Kuka.MovementParameterFieldEnabled=True; ArcTech.WdatVarName=WDAT2; ArcTech.Basic=3.4.3.1264
  ;ENDFOLD
  $BWDSTART = FALSE
  LDAT_ACT = LCPDAT2
  FDAT_ACT = FP4
  BAS(#CP_PARAMS, gArcBasVelDefinition)
  SET_CD_PARAMS (0)
  TRIGGER WHEN PATH = ArcGetPath(#ArcOffBefore, WDAT2) DELAY = 0 DO ArcMainNG(#ArcOffBeforeOffStd, WDAT2, WP4) PRIO = -1
  TRIGGER WHEN PATH = ArcGetPath(#OnTheFlyArcOff, WDAT2) DELAY = 0 DO ArcMainNG(#ArcOffMoveStd, WDAT2, WP4) PRIO = -1
  ArcMainNG(#ArcOffBeforeMoveStd, WDAT2, WP4)
  LIN XP4
  ArcMainNG(#ArcOffAfterMoveStd, WDAT2, WP4)
;ENDFOLD
   $VEL.CP = 0.080
   LIN  {X 8.829, Y 6.566, Z 0.700, A 0.000, B 0.000, C 0.000} C_DIS

;FOLD ARCON WDAT1 LIN P3 Vel=0.5 m/s CPDAT1 Tool[1]:cmttorch Base[1]:vrashatel ;%{PE}
  ;FOLD Parameters ;%{h}
    ;Params IlfProvider=kukaroboter.arctech.arconlin; Kuka.IsGlobalPoint=False; Kuka.PointName=P3; Kuka.BlendingEnabled=False; Kuka.MoveDataName=CPDAT1; Kuka.VelocityPath=0.5; Kuka.CurrentCDSetIndex=0; Kuka.MovementParameterFieldEnabled=True; ArcTech.WdatVarName=WDAT1; ArcTech.Basic=3.4.3.1264
  ;ENDFOLD
  $BWDSTART = FALSE
  LDAT_ACT = LCPDAT1
  FDAT_ACT = FP3
  BAS(#CP_PARAMS, 0.5)
  SET_CD_PARAMS (0)
  TRIGGER WHEN DISTANCE = 1 DELAY = ArcGetDelay(#PreDefinition, WDAT1) DO ArcMainNG(#PreDefinition, WDAT1, WP3) PRIO = -1
  TRIGGER WHEN PATH = ArcGetPath(#OnTheFlyArcOn, WDAT1) DELAY = ArcGetDelay(#GasPreflow, WDAT1) DO ArcMainNG(#GasPreflow, WDAT1, WP3) PRIO = -1
  TRIGGER WHEN PATH = ArcGetPath(#OnTheFlyArcOn, WDAT1) DELAY = 0 DO ArcMainNG(#ArcOnMoveStd, WDAT1, WP3) PRIO = -1
  ArcMainNG(#ArcOnBeforeMoveStd, WDAT1, WP3)
  LIN XP3
  ArcMainNG(#ArcOnAfterMoveStd, WDAT1, WP3)
;ENDFOLD
   $VEL.CP = 0.060
   LIN  {X -6.566, Y -8.829, Z 0.700, A 0.000, B 0.000, C 0.000} C_DIS

;FOLD ARCOFF WDAT2 LIN P4 CPDAT2 Tool[1]:cmttorch Base[1]:vrashatel ;%{PE}
  ;FOLD Parameters ;%{h}
    ;Params IlfProvider=kukaroboter.arctech.arcofflin; Kuka.IsGlobalPoint=False; Kuka.PointName=P4; Kuka.BlendingEnabled=False; Kuka.MoveDataName=CPDAT2; Kuka.VelocityPath=0.01; Kuka.CurrentCDSetIndex=0; Kuka.MovementParameterFieldEnabled=True; ArcTech.WdatVarName=WDAT2; ArcTech.Basic=3.4.3.1264
  ;ENDFOLD
  $BWDSTART = FALSE
  LDAT_ACT = LCPDAT2
  FDAT_ACT = FP4
  BAS(#CP_PARAMS, gArcBasVelDefinition)
  SET_CD_PARAMS (0)
  TRIGGER WHEN PATH = ArcGetPath(#ArcOffBefore, WDAT2) DELAY = 0 DO ArcMainNG(#ArcOffBeforeOffStd, WDAT2, WP4) PRIO = -1
  TRIGGER WHEN PATH = ArcGetPath(#OnTheFlyArcOff, WDAT2) DELAY = 0 DO ArcMainNG(#ArcOffMoveStd, WDAT2, WP4) PRIO = -1
  ArcMainNG(#ArcOffBeforeMoveStd, WDAT2, WP4)
  LIN XP4
  ArcMainNG(#ArcOffAfterMoveStd, WDAT2, WP4)
;ENDFOLD
   $VEL.CP = 0.080
   LIN  {X -6.001, Y -8.829, Z 0.700, A 0.000, B 0.000, C 0.000} C_DIS

;FOLD ARCON WDAT1 LIN P3 Vel=0.5 m/s CPDAT1 Tool[1]:cmttorch Base[1]:vrashatel ;%{PE}
  ;FOLD Parameters ;%{h}
    ;Params IlfProvider=kukaroboter.arctech.arconlin; Kuka.IsGlobalPoint=False; Kuka.PointName=P3; Kuka.BlendingEnabled=False; Kuka.MoveDataName=CPDAT1; Kuka.VelocityPath=0.5; Kuka.CurrentCDSetIndex=0; Kuka.MovementParameterFieldEnabled=True; ArcTech.WdatVarName=WDAT1; ArcTech.Basic=3.4.3.1264
  ;ENDFOLD
  $BWDSTART = FALSE
  LDAT_ACT = LCPDAT1
  FDAT_ACT = FP3
  BAS(#CP_PARAMS, 0.5)
  SET_CD_PARAMS (0)
  TRIGGER WHEN DISTANCE = 1 DELAY = ArcGetDelay(#PreDefinition, WDAT1) DO ArcMainNG(#PreDefinition, WDAT1, WP3) PRIO = -1
  TRIGGER WHEN PATH = ArcGetPath(#OnTheFlyArcOn, WDAT1) DELAY = ArcGetDelay(#GasPreflow, WDAT1) DO ArcMainNG(#GasPreflow, WDAT1, WP3) PRIO = -1
  TRIGGER WHEN PATH = ArcGetPath(#OnTheFlyArcOn, WDAT1) DELAY = 0 DO ArcMainNG(#ArcOnMoveStd, WDAT1, WP3) PRIO = -1
  ArcMainNG(#ArcOnBeforeMoveStd, WDAT1, WP3)
  LIN XP3
  ArcMainNG(#ArcOnAfterMoveStd, WDAT1, WP3)
;ENDFOLD
   $VEL.CP = 0.060
   LIN  {X 8.829, Y 6.001, Z 0.700, A 0.000, B 0.000, C 0.000} C_DIS

;FOLD ARCOFF WDAT2 LIN P4 CPDAT2 Tool[1]:cmttorch Base[1]:vrashatel ;%{PE}
  ;FOLD Parameters ;%{h}
    ;Params IlfProvider=kukaroboter.arctech.arcofflin; Kuka.IsGlobalPoint=False; Kuka.PointName=P4; Kuka.BlendingEnabled=False; Kuka.MoveDataName=CPDAT2; Kuka.VelocityPath=0.01; Kuka.CurrentCDSetIndex=0; Kuka.MovementParameterFieldEnabled=True; ArcTech.WdatVarName=WDAT2; ArcTech.Basic=3.4.3.1264
  ;ENDFOLD
  $BWDSTART = FALSE
  LDAT_ACT = LCPDAT2
  FDAT_ACT = FP4
  BAS(#CP_PARAMS, gArcBasVelDefinition)
  SET_CD_PARAMS (0)
  TRIGGER WHEN PATH = ArcGetPath(#ArcOffBefore, WDAT2) DELAY = 0 DO ArcMainNG(#ArcOffBeforeOffStd, WDAT2, WP4) PRIO = -1
  TRIGGER WHEN PATH = ArcGetPath(#OnTheFlyArcOff, WDAT2) DELAY = 0 DO ArcMainNG(#ArcOffMoveStd, WDAT2, WP4) PRIO = -1
  ArcMainNG(#ArcOffBeforeMoveStd, WDAT2, WP4)
  LIN XP4
  ArcMainNG(#ArcOffAfterMoveStd, WDAT2, WP4)
;ENDFOLD
   $VEL.CP = 0.080
   LIN  {X 8.829, Y 5.435, Z 0.700, A 0.000, B 0.000, C 0.000} C_DIS

;FOLD ARCON WDAT1 LIN P3 Vel=0.5 m/s CPDAT1 Tool[1]:cmttorch Base[1]:vrashatel ;%{PE}
  ;FOLD Parameters ;%{h}
    ;Params IlfProvider=kukaroboter.arctech.arconlin; Kuka.IsGlobalPoint=False; Kuka.PointName=P3; Kuka.BlendingEnabled=False; Kuka.MoveDataName=CPDAT1; Kuka.VelocityPath=0.5; Kuka.CurrentCDSetIndex=0; Kuka.MovementParameterFieldEnabled=True; ArcTech.WdatVarName=WDAT1; ArcTech.Basic=3.4.3.1264
  ;ENDFOLD
  $BWDSTART = FALSE
  LDAT_ACT = LCPDAT1
  FDAT_ACT = FP3
  BAS(#CP_PARAMS, 0.5)
  SET_CD_PARAMS (0)
  TRIGGER WHEN DISTANCE = 1 DELAY = ArcGetDelay(#PreDefinition, WDAT1) DO ArcMainNG(#PreDefinition, WDAT1, WP3) PRIO = -1
  TRIGGER WHEN PATH = ArcGetPath(#OnTheFlyArcOn, WDAT1) DELAY = ArcGetDelay(#GasPreflow, WDAT1) DO ArcMainNG(#GasPreflow, WDAT1, WP3) PRIO = -1
  TRIGGER WHEN PATH = ArcGetPath(#OnTheFlyArcOn, WDAT1) DELAY = 0 DO ArcMainNG(#ArcOnMoveStd, WDAT1, WP3) PRIO = -1
  ArcMainNG(#ArcOnBeforeMoveStd, WDAT1, WP3)
  LIN XP3
  ArcMainNG(#ArcOnAfterMoveStd, WDAT1, WP3)
;ENDFOLD
   $VEL.CP = 0.060
   LIN  {X -5.435, Y -8.829, Z 0.700, A 0.000, B 0.000, C 0.000} C_DIS

;FOLD ARCOFF WDAT2 LIN P4 CPDAT2 Tool[1]:cmttorch Base[1]:vrashatel ;%{PE}
  ;FOLD Parameters ;%{h}
    ;Params IlfProvider=kukaroboter.arctech.arcofflin; Kuka.IsGlobalPoint=False; Kuka.PointName=P4; Kuka.BlendingEnabled=False; Kuka.MoveDataName=CPDAT2; Kuka.VelocityPath=0.01; Kuka.CurrentCDSetIndex=0; Kuka.MovementParameterFieldEnabled=True; ArcTech.WdatVarName=WDAT2; ArcTech.Basic=3.4.3.1264
  ;ENDFOLD
  $BWDSTART = FALSE
  LDAT_ACT = LCPDAT2
  FDAT_ACT = FP4
  BAS(#CP_PARAMS, gArcBasVelDefinition)
  SET_CD_PARAMS (0)
  TRIGGER WHEN PATH = ArcGetPath(#ArcOffBefore, WDAT2) DELAY = 0 DO ArcMainNG(#ArcOffBeforeOffStd, WDAT2, WP4) PRIO = -1
  TRIGGER WHEN PATH = ArcGetPath(#OnTheFlyArcOff, WDAT2) DELAY = 0 DO ArcMainNG(#ArcOffMoveStd, WDAT2, WP4) PRIO = -1
  ArcMainNG(#ArcOffBeforeMoveStd, WDAT2, WP4)
  LIN XP4
  ArcMainNG(#ArcOffAfterMoveStd, WDAT2, WP4)
;ENDFOLD
   $VEL.CP = 0.080
   LIN  {X -4.869, Y -8.829, Z 0.700, A 0.000, B 0.000, C 0.000} C_DIS

;FOLD ARCON WDAT1 LIN P3 Vel=0.5 m/s CPDAT1 Tool[1]:cmttorch Base[1]:vrashatel ;%{PE}
  ;FOLD Parameters ;%{h}
    ;Params IlfProvider=kukaroboter.arctech.arconlin; Kuka.IsGlobalPoint=False; Kuka.PointName=P3; Kuka.BlendingEnabled=False; Kuka.MoveDataName=CPDAT1; Kuka.VelocityPath=0.5; Kuka.CurrentCDSetIndex=0; Kuka.MovementParameterFieldEnabled=True; ArcTech.WdatVarName=WDAT1; ArcTech.Basic=3.4.3.1264
  ;ENDFOLD
  $BWDSTART = FALSE
  LDAT_ACT = LCPDAT1
  FDAT_ACT = FP3
  BAS(#CP_PARAMS, 0.5)
  SET_CD_PARAMS (0)
  TRIGGER WHEN DISTANCE = 1 DELAY = ArcGetDelay(#PreDefinition, WDAT1) DO ArcMainNG(#PreDefinition, WDAT1, WP3) PRIO = -1
  TRIGGER WHEN PATH = ArcGetPath(#OnTheFlyArcOn, WDAT1) DELAY = ArcGetDelay(#GasPreflow, WDAT1) DO ArcMainNG(#GasPreflow, WDAT1, WP3) PRIO = -1
  TRIGGER WHEN PATH = ArcGetPath(#OnTheFlyArcOn, WDAT1) DELAY = 0 DO ArcMainNG(#ArcOnMoveStd, WDAT1, WP3) PRIO = -1
  ArcMainNG(#ArcOnBeforeMoveStd, WDAT1, WP3)
  LIN XP3
  ArcMainNG(#ArcOnAfterMoveStd, WDAT1, WP3)
;ENDFOLD
   $VEL.CP = 0.060
   LIN  {X 8.829, Y 4.869, Z 0.700, A 0.000, B 0.000, C 0.000} C_DIS

;FOLD ARCOFF WDAT2 LIN P4 CPDAT2 Tool[1]:cmttorch Base[1]:vrashatel ;%{PE}
  ;FOLD Parameters ;%{h}
    ;Params IlfProvider=kukaroboter.arctech.arcofflin; Kuka.IsGlobalPoint=False; Kuka.PointName=P4; Kuka.BlendingEnabled=False; Kuka.MoveDataName=CPDAT2; Kuka.VelocityPath=0.01; Kuka.CurrentCDSetIndex=0; Kuka.MovementParameterFieldEnabled=True; ArcTech.WdatVarName=WDAT2; ArcTech.Basic=3.4.3.1264
  ;ENDFOLD
  $BWDSTART = FALSE
  LDAT_ACT = LCPDAT2
  FDAT_ACT = FP4
  BAS(#CP_PARAMS, gArcBasVelDefinition)
  SET_CD_PARAMS (0)
  TRIGGER WHEN PATH = ArcGetPath(#ArcOffBefore, WDAT2) DELAY = 0 DO ArcMainNG(#ArcOffBeforeOffStd, WDAT2, WP4) PRIO = -1
  TRIGGER WHEN PATH = ArcGetPath(#OnTheFlyArcOff, WDAT2) DELAY = 0 DO ArcMainNG(#ArcOffMoveStd, WDAT2, WP4) PRIO = -1
  ArcMainNG(#ArcOffBeforeMoveStd, WDAT2, WP4)
  LIN XP4
  ArcMainNG(#ArcOffAfterMoveStd, WDAT2, WP4)
;ENDFOLD
   $VEL.CP = 0.080
   LIN  {X 8.829, Y 4.304, Z 0.700, A 0.000, B 0.000, C 0.000} C_DIS

;FOLD ARCON WDAT1 LIN P3 Vel=0.5 m/s CPDAT1 Tool[1]:cmttorch Base[1]:vrashatel ;%{PE}
  ;FOLD Parameters ;%{h}
    ;Params IlfProvider=kukaroboter.arctech.arconlin; Kuka.IsGlobalPoint=False; Kuka.PointName=P3; Kuka.BlendingEnabled=False; Kuka.MoveDataName=CPDAT1; Kuka.VelocityPath=0.5; Kuka.CurrentCDSetIndex=0; Kuka.MovementParameterFieldEnabled=True; ArcTech.WdatVarName=WDAT1; ArcTech.Basic=3.4.3.1264
  ;ENDFOLD
  $BWDSTART = FALSE
  LDAT_ACT = LCPDAT1
  FDAT_ACT = FP3
  BAS(#CP_PARAMS, 0.5)
  SET_CD_PARAMS (0)
  TRIGGER WHEN DISTANCE = 1 DELAY = ArcGetDelay(#PreDefinition, WDAT1) DO ArcMainNG(#PreDefinition, WDAT1, WP3) PRIO = -1
  TRIGGER WHEN PATH = ArcGetPath(#OnTheFlyArcOn, WDAT1) DELAY = ArcGetDelay(#GasPreflow, WDAT1) DO ArcMainNG(#GasPreflow, WDAT1, WP3) PRIO = -1
  TRIGGER WHEN PATH = ArcGetPath(#OnTheFlyArcOn, WDAT1) DELAY = 0 DO ArcMainNG(#ArcOnMoveStd, WDAT1, WP3) PRIO = -1
  ArcMainNG(#ArcOnBeforeMoveStd, WDAT1, WP3)
  LIN XP3
  ArcMainNG(#ArcOnAfterMoveStd, WDAT1, WP3)
;ENDFOLD
   $VEL.CP = 0.060
   LIN  {X -4.304, Y -8.829, Z 0.700, A 0.000, B 0.000, C 0.000} C_DIS

;FOLD ARCOFF WDAT2 LIN P4 CPDAT2 Tool[1]:cmttorch Base[1]:vrashatel ;%{PE}
  ;FOLD Parameters ;%{h}
    ;Params IlfProvider=kukaroboter.arctech.arcofflin; Kuka.IsGlobalPoint=False; Kuka.PointName=P4; Kuka.BlendingEnabled=False; Kuka.MoveDataName=CPDAT2; Kuka.VelocityPath=0.01; Kuka.CurrentCDSetIndex=0; Kuka.MovementParameterFieldEnabled=True; ArcTech.WdatVarName=WDAT2; ArcTech.Basic=3.4.3.1264
  ;ENDFOLD
  $BWDSTART = FALSE
  LDAT_ACT = LCPDAT2
  FDAT_ACT = FP4
  BAS(#CP_PARAMS, gArcBasVelDefinition)
  SET_CD_PARAMS (0)
  TRIGGER WHEN PATH = ArcGetPath(#ArcOffBefore, WDAT2) DELAY = 0 DO ArcMainNG(#ArcOffBeforeOffStd, WDAT2, WP4) PRIO = -1
  TRIGGER WHEN PATH = ArcGetPath(#OnTheFlyArcOff, WDAT2) DELAY = 0 DO ArcMainNG(#ArcOffMoveStd, WDAT2, WP4) PRIO = -1
  ArcMainNG(#ArcOffBeforeMoveStd, WDAT2, WP4)
  LIN XP4
  ArcMainNG(#ArcOffAfterMoveStd, WDAT2, WP4)
;ENDFOLD
   $VEL.CP = 0.080
   LIN  {X -3.738, Y -8.829, Z 0.700, A 0.000, B 0.000, C 0.000} C_DIS

;FOLD ARCON WDAT1 LIN P3 Vel=0.5 m/s CPDAT1 Tool[1]:cmttorch Base[1]:vrashatel ;%{PE}
  ;FOLD Parameters ;%{h}
    ;Params IlfProvider=kukaroboter.arctech.arconlin; Kuka.IsGlobalPoint=False; Kuka.PointName=P3; Kuka.BlendingEnabled=False; Kuka.MoveDataName=CPDAT1; Kuka.VelocityPath=0.5; Kuka.CurrentCDSetIndex=0; Kuka.MovementParameterFieldEnabled=True; ArcTech.WdatVarName=WDAT1; ArcTech.Basic=3.4.3.1264
  ;ENDFOLD
  $BWDSTART = FALSE
  LDAT_ACT = LCPDAT1
  FDAT_ACT = FP3
  BAS(#CP_PARAMS, 0.5)
  SET_CD_PARAMS (0)
  TRIGGER WHEN DISTANCE = 1 DELAY = ArcGetDelay(#PreDefinition, WDAT1) DO ArcMainNG(#PreDefinition, WDAT1, WP3) PRIO = -1
  TRIGGER WHEN PATH = ArcGetPath(#OnTheFlyArcOn, WDAT1) DELAY = ArcGetDelay(#GasPreflow, WDAT1) DO ArcMainNG(#GasPreflow, WDAT1, WP3) PRIO = -1
  TRIGGER WHEN PATH = ArcGetPath(#OnTheFlyArcOn, WDAT1) DELAY = 0 DO ArcMainNG(#ArcOnMoveStd, WDAT1, WP3) PRIO = -1
  ArcMainNG(#ArcOnBeforeMoveStd, WDAT1, WP3)
  LIN XP3
  ArcMainNG(#ArcOnAfterMoveStd, WDAT1, WP3)
;ENDFOLD
   $VEL.CP = 0.060
   LIN  {X 8.829, Y 3.738, Z 0.700, A 0.000, B 0.000, C 0.000} C_DIS

;FOLD ARCOFF WDAT2 LIN P4 CPDAT2 Tool[1]:cmttorch Base[1]:vrashatel ;%{PE}
  ;FOLD Parameters ;%{h}
    ;Params IlfProvider=kukaroboter.arctech.arcofflin; Kuka.IsGlobalPoint=False; Kuka.PointName=P4; Kuka.BlendingEnabled=False; Kuka.MoveDataName=CPDAT2; Kuka.VelocityPath=0.01; Kuka.CurrentCDSetIndex=0; Kuka.MovementParameterFieldEnabled=True; ArcTech.WdatVarName=WDAT2; ArcTech.Basic=3.4.3.1264
  ;ENDFOLD
  $BWDSTART = FALSE
  LDAT_ACT = LCPDAT2
  FDAT_ACT = FP4
  BAS(#CP_PARAMS, gArcBasVelDefinition)
  SET_CD_PARAMS (0)
  TRIGGER WHEN PATH = ArcGetPath(#ArcOffBefore, WDAT2) DELAY = 0 DO ArcMainNG(#ArcOffBeforeOffStd, WDAT2, WP4) PRIO = -1
  TRIGGER WHEN PATH = ArcGetPath(#OnTheFlyArcOff, WDAT2) DELAY = 0 DO ArcMainNG(#ArcOffMoveStd, WDAT2, WP4) PRIO = -1
  ArcMainNG(#ArcOffBeforeMoveStd, WDAT2, WP4)
  LIN XP4
  ArcMainNG(#ArcOffAfterMoveStd, WDAT2, WP4)
;ENDFOLD
   $VEL.CP = 0.080
   LIN  {X 8.829, Y 3.172, Z 0.700, A 0.000, B 0.000, C 0.000} C_DIS

;FOLD ARCON WDAT1 LIN P3 Vel=0.5 m/s CPDAT1 Tool[1]:cmttorch Base[1]:vrashatel ;%{PE}
  ;FOLD Parameters ;%{h}
    ;Params IlfProvider=kukaroboter.arctech.arconlin; Kuka.IsGlobalPoint=False; Kuka.PointName=P3; Kuka.BlendingEnabled=False; Kuka.MoveDataName=CPDAT1; Kuka.VelocityPath=0.5; Kuka.CurrentCDSetIndex=0; Kuka.MovementParameterFieldEnabled=True; ArcTech.WdatVarName=WDAT1; ArcTech.Basic=3.4.3.1264
  ;ENDFOLD
  $BWDSTART = FALSE
  LDAT_ACT = LCPDAT1
  FDAT_ACT = FP3
  BAS(#CP_PARAMS, 0.5)
  SET_CD_PARAMS (0)
  TRIGGER WHEN DISTANCE = 1 DELAY = ArcGetDelay(#PreDefinition, WDAT1) DO ArcMainNG(#PreDefinition, WDAT1, WP3) PRIO = -1
  TRIGGER WHEN PATH = ArcGetPath(#OnTheFlyArcOn, WDAT1) DELAY = ArcGetDelay(#GasPreflow, WDAT1) DO ArcMainNG(#GasPreflow, WDAT1, WP3) PRIO = -1
  TRIGGER WHEN PATH = ArcGetPath(#OnTheFlyArcOn, WDAT1) DELAY = 0 DO ArcMainNG(#ArcOnMoveStd, WDAT1, WP3) PRIO = -1
  ArcMainNG(#ArcOnBeforeMoveStd, WDAT1, WP3)
  LIN XP3
  ArcMainNG(#ArcOnAfterMoveStd, WDAT1, WP3)
;ENDFOLD
   $VEL.CP = 0.060
   LIN  {X -3.172, Y -8.829, Z 0.700, A 0.000, B 0.000, C 0.000} C_DIS

;FOLD ARCOFF WDAT2 LIN P4 CPDAT2 Tool[1]:cmttorch Base[1]:vrashatel ;%{PE}
  ;FOLD Parameters ;%{h}
    ;Params IlfProvider=kukaroboter.arctech.arcofflin; Kuka.IsGlobalPoint=False; Kuka.PointName=P4; Kuka.BlendingEnabled=False; Kuka.MoveDataName=CPDAT2; Kuka.VelocityPath=0.01; Kuka.CurrentCDSetIndex=0; Kuka.MovementParameterFieldEnabled=True; ArcTech.WdatVarName=WDAT2; ArcTech.Basic=3.4.3.1264
  ;ENDFOLD
  $BWDSTART = FALSE
  LDAT_ACT = LCPDAT2
  FDAT_ACT = FP4
  BAS(#CP_PARAMS, gArcBasVelDefinition)
  SET_CD_PARAMS (0)
  TRIGGER WHEN PATH = ArcGetPath(#ArcOffBefore, WDAT2) DELAY = 0 DO ArcMainNG(#ArcOffBeforeOffStd, WDAT2, WP4) PRIO = -1
  TRIGGER WHEN PATH = ArcGetPath(#OnTheFlyArcOff, WDAT2) DELAY = 0 DO ArcMainNG(#ArcOffMoveStd, WDAT2, WP4) PRIO = -1
  ArcMainNG(#ArcOffBeforeMoveStd, WDAT2, WP4)
  LIN XP4
  ArcMainNG(#ArcOffAfterMoveStd, WDAT2, WP4)
;ENDFOLD
   $VEL.CP = 0.080
   LIN  {X -2.607, Y -8.829, Z 0.700, A 0.000, B 0.000, C 0.000} C_DIS

;FOLD ARCON WDAT1 LIN P3 Vel=0.5 m/s CPDAT1 Tool[1]:cmttorch Base[1]:vrashatel ;%{PE}
  ;FOLD Parameters ;%{h}
    ;Params IlfProvider=kukaroboter.arctech.arconlin; Kuka.IsGlobalPoint=False; Kuka.PointName=P3; Kuka.BlendingEnabled=False; Kuka.MoveDataName=CPDAT1; Kuka.VelocityPath=0.5; Kuka.CurrentCDSetIndex=0; Kuka.MovementParameterFieldEnabled=True; ArcTech.WdatVarName=WDAT1; ArcTech.Basic=3.4.3.1264
  ;ENDFOLD
  $BWDSTART = FALSE
  LDAT_ACT = LCPDAT1
  FDAT_ACT = FP3
  BAS(#CP_PARAMS, 0.5)
  SET_CD_PARAMS (0)
  TRIGGER WHEN DISTANCE = 1 DELAY = ArcGetDelay(#PreDefinition, WDAT1) DO ArcMainNG(#PreDefinition, WDAT1, WP3) PRIO = -1
  TRIGGER WHEN PATH = ArcGetPath(#OnTheFlyArcOn, WDAT1) DELAY = ArcGetDelay(#GasPreflow, WDAT1) DO ArcMainNG(#GasPreflow, WDAT1, WP3) PRIO = -1
  TRIGGER WHEN PATH = ArcGetPath(#OnTheFlyArcOn, WDAT1) DELAY = 0 DO ArcMainNG(#ArcOnMoveStd, WDAT1, WP3) PRIO = -1
  ArcMainNG(#ArcOnBeforeMoveStd, WDAT1, WP3)
  LIN XP3
  ArcMainNG(#ArcOnAfterMoveStd, WDAT1, WP3)
;ENDFOLD
   $VEL.CP = 0.060
   LIN  {X 8.829, Y 2.607, Z 0.700, A 0.000, B 0.000, C 0.000} C_DIS

;FOLD ARCOFF WDAT2 LIN P4 CPDAT2 Tool[1]:cmttorch Base[1]:vrashatel ;%{PE}
  ;FOLD Parameters ;%{h}
    ;Params IlfProvider=kukaroboter.arctech.arcofflin; Kuka.IsGlobalPoint=False; Kuka.PointName=P4; Kuka.BlendingEnabled=False; Kuka.MoveDataName=CPDAT2; Kuka.VelocityPath=0.01; Kuka.CurrentCDSetIndex=0; Kuka.MovementParameterFieldEnabled=True; ArcTech.WdatVarName=WDAT2; ArcTech.Basic=3.4.3.1264
  ;ENDFOLD
  $BWDSTART = FALSE
  LDAT_ACT = LCPDAT2
  FDAT_ACT = FP4
  BAS(#CP_PARAMS, gArcBasVelDefinition)
  SET_CD_PARAMS (0)
  TRIGGER WHEN PATH = ArcGetPath(#ArcOffBefore, WDAT2) DELAY = 0 DO ArcMainNG(#ArcOffBeforeOffStd, WDAT2, WP4) PRIO = -1
  TRIGGER WHEN PATH = ArcGetPath(#OnTheFlyArcOff, WDAT2) DELAY = 0 DO ArcMainNG(#ArcOffMoveStd, WDAT2, WP4) PRIO = -1
  ArcMainNG(#ArcOffBeforeMoveStd, WDAT2, WP4)
  LIN XP4
  ArcMainNG(#ArcOffAfterMoveStd, WDAT2, WP4)
;ENDFOLD
   $VEL.CP = 0.080
   LIN  {X 8.829, Y 2.041, Z 0.700, A 0.000, B 0.000, C 0.000} C_DIS

;FOLD ARCON WDAT1 LIN P3 Vel=0.5 m/s CPDAT1 Tool[1]:cmttorch Base[1]:vrashatel ;%{PE}
  ;FOLD Parameters ;%{h}
    ;Params IlfProvider=kukaroboter.arctech.arconlin; Kuka.IsGlobalPoint=False; Kuka.PointName=P3; Kuka.BlendingEnabled=False; Kuka.MoveDataName=CPDAT1; Kuka.VelocityPath=0.5; Kuka.CurrentCDSetIndex=0; Kuka.MovementParameterFieldEnabled=True; ArcTech.WdatVarName=WDAT1; ArcTech.Basic=3.4.3.1264
  ;ENDFOLD
  $BWDSTART = FALSE
  LDAT_ACT = LCPDAT1
  FDAT_ACT = FP3
  BAS(#CP_PARAMS, 0.5)
  SET_CD_PARAMS (0)
  TRIGGER WHEN DISTANCE = 1 DELAY = ArcGetDelay(#PreDefinition, WDAT1) DO ArcMainNG(#PreDefinition, WDAT1, WP3) PRIO = -1
  TRIGGER WHEN PATH = ArcGetPath(#OnTheFlyArcOn, WDAT1) DELAY = ArcGetDelay(#GasPreflow, WDAT1) DO ArcMainNG(#GasPreflow, WDAT1, WP3) PRIO = -1
  TRIGGER WHEN PATH = ArcGetPath(#OnTheFlyArcOn, WDAT1) DELAY = 0 DO ArcMainNG(#ArcOnMoveStd, WDAT1, WP3) PRIO = -1
  ArcMainNG(#ArcOnBeforeMoveStd, WDAT1, WP3)
  LIN XP3
  ArcMainNG(#ArcOnAfterMoveStd, WDAT1, WP3)
;ENDFOLD
   $VEL.CP = 0.060
   LIN  {X -2.041, Y -8.829, Z 0.700, A 0.000, B 0.000, C 0.000} C_DIS

;FOLD ARCOFF WDAT2 LIN P4 CPDAT2 Tool[1]:cmttorch Base[1]:vrashatel ;%{PE}
  ;FOLD Parameters ;%{h}
    ;Params IlfProvider=kukaroboter.arctech.arcofflin; Kuka.IsGlobalPoint=False; Kuka.PointName=P4; Kuka.BlendingEnabled=False; Kuka.MoveDataName=CPDAT2; Kuka.VelocityPath=0.01; Kuka.CurrentCDSetIndex=0; Kuka.MovementParameterFieldEnabled=True; ArcTech.WdatVarName=WDAT2; ArcTech.Basic=3.4.3.1264
  ;ENDFOLD
  $BWDSTART = FALSE
  LDAT_ACT = LCPDAT2
  FDAT_ACT = FP4
  BAS(#CP_PARAMS, gArcBasVelDefinition)
  SET_CD_PARAMS (0)
  TRIGGER WHEN PATH = ArcGetPath(#ArcOffBefore, WDAT2) DELAY = 0 DO ArcMainNG(#ArcOffBeforeOffStd, WDAT2, WP4) PRIO = -1
  TRIGGER WHEN PATH = ArcGetPath(#OnTheFlyArcOff, WDAT2) DELAY = 0 DO ArcMainNG(#ArcOffMoveStd, WDAT2, WP4) PRIO = -1
  ArcMainNG(#ArcOffBeforeMoveStd, WDAT2, WP4)
  LIN XP4
  ArcMainNG(#ArcOffAfterMoveStd, WDAT2, WP4)
;ENDFOLD
   $VEL.CP = 0.080
   LIN  {X -1.475, Y -8.829, Z 0.700, A 0.000, B 0.000, C 0.000} C_DIS

;FOLD ARCON WDAT1 LIN P3 Vel=0.5 m/s CPDAT1 Tool[1]:cmttorch Base[1]:vrashatel ;%{PE}
  ;FOLD Parameters ;%{h}
    ;Params IlfProvider=kukaroboter.arctech.arconlin; Kuka.IsGlobalPoint=False; Kuka.PointName=P3; Kuka.BlendingEnabled=False; Kuka.MoveDataName=CPDAT1; Kuka.VelocityPath=0.5; Kuka.CurrentCDSetIndex=0; Kuka.MovementParameterFieldEnabled=True; ArcTech.WdatVarName=WDAT1; ArcTech.Basic=3.4.3.1264
  ;ENDFOLD
  $BWDSTART = FALSE
  LDAT_ACT = LCPDAT1
  FDAT_ACT = FP3
  BAS(#CP_PARAMS, 0.5)
  SET_CD_PARAMS (0)
  TRIGGER WHEN DISTANCE = 1 DELAY = ArcGetDelay(#PreDefinition, WDAT1) DO ArcMainNG(#PreDefinition, WDAT1, WP3) PRIO = -1
  TRIGGER WHEN PATH = ArcGetPath(#OnTheFlyArcOn, WDAT1) DELAY = ArcGetDelay(#GasPreflow, WDAT1) DO ArcMainNG(#GasPreflow, WDAT1, WP3) PRIO = -1
  TRIGGER WHEN PATH = ArcGetPath(#OnTheFlyArcOn, WDAT1) DELAY = 0 DO ArcMainNG(#ArcOnMoveStd, WDAT1, WP3) PRIO = -1
  ArcMainNG(#ArcOnBeforeMoveStd, WDAT1, WP3)
  LIN XP3
  ArcMainNG(#ArcOnAfterMoveStd, WDAT1, WP3)
;ENDFOLD
   $VEL.CP = 0.060
   LIN  {X 8.829, Y 1.475, Z 0.700, A 0.000, B 0.000, C 0.000} C_DIS

;FOLD ARCOFF WDAT2 LIN P4 CPDAT2 Tool[1]:cmttorch Base[1]:vrashatel ;%{PE}
  ;FOLD Parameters ;%{h}
    ;Params IlfProvider=kukaroboter.arctech.arcofflin; Kuka.IsGlobalPoint=False; Kuka.PointName=P4; Kuka.BlendingEnabled=False; Kuka.MoveDataName=CPDAT2; Kuka.VelocityPath=0.01; Kuka.CurrentCDSetIndex=0; Kuka.MovementParameterFieldEnabled=True; ArcTech.WdatVarName=WDAT2; ArcTech.Basic=3.4.3.1264
  ;ENDFOLD
  $BWDSTART = FALSE
  LDAT_ACT = LCPDAT2
  FDAT_ACT = FP4
  BAS(#CP_PARAMS, gArcBasVelDefinition)
  SET_CD_PARAMS (0)
  TRIGGER WHEN PATH = ArcGetPath(#ArcOffBefore, WDAT2) DELAY = 0 DO ArcMainNG(#ArcOffBeforeOffStd, WDAT2, WP4) PRIO = -1
  TRIGGER WHEN PATH = ArcGetPath(#OnTheFlyArcOff, WDAT2) DELAY = 0 DO ArcMainNG(#ArcOffMoveStd, WDAT2, WP4) PRIO = -1
  ArcMainNG(#ArcOffBeforeMoveStd, WDAT2, WP4)
  LIN XP4
  ArcMainNG(#ArcOffAfterMoveStd, WDAT2, WP4)
;ENDFOLD
   $VEL.CP = 0.080
   LIN  {X 8.829, Y 0.910, Z 0.700, A 0.000, B 0.000, C 0.000} C_DIS

;FOLD ARCON WDAT1 LIN P3 Vel=0.5 m/s CPDAT1 Tool[1]:cmttorch Base[1]:vrashatel ;%{PE}
  ;FOLD Parameters ;%{h}
    ;Params IlfProvider=kukaroboter.arctech.arconlin; Kuka.IsGlobalPoint=False; Kuka.PointName=P3; Kuka.BlendingEnabled=False; Kuka.MoveDataName=CPDAT1; Kuka.VelocityPath=0.5; Kuka.CurrentCDSetIndex=0; Kuka.MovementParameterFieldEnabled=True; ArcTech.WdatVarName=WDAT1; ArcTech.Basic=3.4.3.1264
  ;ENDFOLD
  $BWDSTART = FALSE
  LDAT_ACT = LCPDAT1
  FDAT_ACT = FP3
  BAS(#CP_PARAMS, 0.5)
  SET_CD_PARAMS (0)
  TRIGGER WHEN DISTANCE = 1 DELAY = ArcGetDelay(#PreDefinition, WDAT1) DO ArcMainNG(#PreDefinition, WDAT1, WP3) PRIO = -1
  TRIGGER WHEN PATH = ArcGetPath(#OnTheFlyArcOn, WDAT1) DELAY = ArcGetDelay(#GasPreflow, WDAT1) DO ArcMainNG(#GasPreflow, WDAT1, WP3) PRIO = -1
  TRIGGER WHEN PATH = ArcGetPath(#OnTheFlyArcOn, WDAT1) DELAY = 0 DO ArcMainNG(#ArcOnMoveStd, WDAT1, WP3) PRIO = -1
  ArcMainNG(#ArcOnBeforeMoveStd, WDAT1, WP3)
  LIN XP3
  ArcMainNG(#ArcOnAfterMoveStd, WDAT1, WP3)
;ENDFOLD
   $VEL.CP = 0.060
   LIN  {X -0.910, Y -8.829, Z 0.700, A 0.000, B 0.000, C 0.000} C_DIS

;FOLD ARCOFF WDAT2 LIN P4 CPDAT2 Tool[1]:cmttorch Base[1]:vrashatel ;%{PE}
  ;FOLD Parameters ;%{h}
    ;Params IlfProvider=kukaroboter.arctech.arcofflin; Kuka.IsGlobalPoint=False; Kuka.PointName=P4; Kuka.BlendingEnabled=False; Kuka.MoveDataName=CPDAT2; Kuka.VelocityPath=0.01; Kuka.CurrentCDSetIndex=0; Kuka.MovementParameterFieldEnabled=True; ArcTech.WdatVarName=WDAT2; ArcTech.Basic=3.4.3.1264
  ;ENDFOLD
  $BWDSTART = FALSE
  LDAT_ACT = LCPDAT2
  FDAT_ACT = FP4
  BAS(#CP_PARAMS, gArcBasVelDefinition)
  SET_CD_PARAMS (0)
  TRIGGER WHEN PATH = ArcGetPath(#ArcOffBefore, WDAT2) DELAY = 0 DO ArcMainNG(#ArcOffBeforeOffStd, WDAT2, WP4) PRIO = -1
  TRIGGER WHEN PATH = ArcGetPath(#OnTheFlyArcOff, WDAT2) DELAY = 0 DO ArcMainNG(#ArcOffMoveStd, WDAT2, WP4) PRIO = -1
  ArcMainNG(#ArcOffBeforeMoveStd, WDAT2, WP4)
  LIN XP4
  ArcMainNG(#ArcOffAfterMoveStd, WDAT2, WP4)
;ENDFOLD
   $VEL.CP = 0.080
   LIN  {X -0.344, Y -8.829, Z 0.700, A 0.000, B 0.000, C 0.000} C_DIS

;FOLD ARCON WDAT1 LIN P3 Vel=0.5 m/s CPDAT1 Tool[1]:cmttorch Base[1]:vrashatel ;%{PE}
  ;FOLD Parameters ;%{h}
    ;Params IlfProvider=kukaroboter.arctech.arconlin; Kuka.IsGlobalPoint=False; Kuka.PointName=P3; Kuka.BlendingEnabled=False; Kuka.MoveDataName=CPDAT1; Kuka.VelocityPath=0.5; Kuka.CurrentCDSetIndex=0; Kuka.MovementParameterFieldEnabled=True; ArcTech.WdatVarName=WDAT1; ArcTech.Basic=3.4.3.1264
  ;ENDFOLD
  $BWDSTART = FALSE
  LDAT_ACT = LCPDAT1
  FDAT_ACT = FP3
  BAS(#CP_PARAMS, 0.5)
  SET_CD_PARAMS (0)
  TRIGGER WHEN DISTANCE = 1 DELAY = ArcGetDelay(#PreDefinition, WDAT1) DO ArcMainNG(#PreDefinition, WDAT1, WP3) PRIO = -1
  TRIGGER WHEN PATH = ArcGetPath(#OnTheFlyArcOn, WDAT1) DELAY = ArcGetDelay(#GasPreflow, WDAT1) DO ArcMainNG(#GasPreflow, WDAT1, WP3) PRIO = -1
  TRIGGER WHEN PATH = ArcGetPath(#OnTheFlyArcOn, WDAT1) DELAY = 0 DO ArcMainNG(#ArcOnMoveStd, WDAT1, WP3) PRIO = -1
  ArcMainNG(#ArcOnBeforeMoveStd, WDAT1, WP3)
  LIN XP3
  ArcMainNG(#ArcOnAfterMoveStd, WDAT1, WP3)
;ENDFOLD
   $VEL.CP = 0.060
   LIN  {X 8.829, Y 0.344, Z 0.700, A 0.000, B 0.000, C 0.000} C_DIS

;FOLD ARCOFF WDAT2 LIN P4 CPDAT2 Tool[1]:cmttorch Base[1]:vrashatel ;%{PE}
  ;FOLD Parameters ;%{h}
    ;Params IlfProvider=kukaroboter.arctech.arcofflin; Kuka.IsGlobalPoint=False; Kuka.PointName=P4; Kuka.BlendingEnabled=False; Kuka.MoveDataName=CPDAT2; Kuka.VelocityPath=0.01; Kuka.CurrentCDSetIndex=0; Kuka.MovementParameterFieldEnabled=True; ArcTech.WdatVarName=WDAT2; ArcTech.Basic=3.4.3.1264
  ;ENDFOLD
  $BWDSTART = FALSE
  LDAT_ACT = LCPDAT2
  FDAT_ACT = FP4
  BAS(#CP_PARAMS, gArcBasVelDefinition)
  SET_CD_PARAMS (0)
  TRIGGER WHEN PATH = ArcGetPath(#ArcOffBefore, WDAT2) DELAY = 0 DO ArcMainNG(#ArcOffBeforeOffStd, WDAT2, WP4) PRIO = -1
  TRIGGER WHEN PATH = ArcGetPath(#OnTheFlyArcOff, WDAT2) DELAY = 0 DO ArcMainNG(#ArcOffMoveStd, WDAT2, WP4) PRIO = -1
  ArcMainNG(#ArcOffBeforeMoveStd, WDAT2, WP4)
  LIN XP4
  ArcMainNG(#ArcOffAfterMoveStd, WDAT2, WP4)
;ENDFOLD
   $VEL.CP = 0.080
   LIN  {X 8.829, Y -0.221, Z 0.700, A 0.000, B 0.000, C 0.000} C_DIS

;FOLD ARCON WDAT1 LIN P3 Vel=0.5 m/s CPDAT1 Tool[1]:cmttorch Base[1]:vrashatel ;%{PE}
  ;FOLD Parameters ;%{h}
    ;Params IlfProvider=kukaroboter.arctech.arconlin; Kuka.IsGlobalPoint=False; Kuka.PointName=P3; Kuka.BlendingEnabled=False; Kuka.MoveDataName=CPDAT1; Kuka.VelocityPath=0.5; Kuka.CurrentCDSetIndex=0; Kuka.MovementParameterFieldEnabled=True; ArcTech.WdatVarName=WDAT1; ArcTech.Basic=3.4.3.1264
  ;ENDFOLD
  $BWDSTART = FALSE
  LDAT_ACT = LCPDAT1
  FDAT_ACT = FP3
  BAS(#CP_PARAMS, 0.5)
  SET_CD_PARAMS (0)
  TRIGGER WHEN DISTANCE = 1 DELAY = ArcGetDelay(#PreDefinition, WDAT1) DO ArcMainNG(#PreDefinition, WDAT1, WP3) PRIO = -1
  TRIGGER WHEN PATH = ArcGetPath(#OnTheFlyArcOn, WDAT1) DELAY = ArcGetDelay(#GasPreflow, WDAT1) DO ArcMainNG(#GasPreflow, WDAT1, WP3) PRIO = -1
  TRIGGER WHEN PATH = ArcGetPath(#OnTheFlyArcOn, WDAT1) DELAY = 0 DO ArcMainNG(#ArcOnMoveStd, WDAT1, WP3) PRIO = -1
  ArcMainNG(#ArcOnBeforeMoveStd, WDAT1, WP3)
  LIN XP3
  ArcMainNG(#ArcOnAfterMoveStd, WDAT1, WP3)
;ENDFOLD
   $VEL.CP = 0.060
   LIN  {X 0.221, Y -8.829, Z 0.700, A 0.000, B 0.000, C 0.000} C_DIS

;FOLD ARCOFF WDAT2 LIN P4 CPDAT2 Tool[1]:cmttorch Base[1]:vrashatel ;%{PE}
  ;FOLD Parameters ;%{h}
    ;Params IlfProvider=kukaroboter.arctech.arcofflin; Kuka.IsGlobalPoint=False; Kuka.PointName=P4; Kuka.BlendingEnabled=False; Kuka.MoveDataName=CPDAT2; Kuka.VelocityPath=0.01; Kuka.CurrentCDSetIndex=0; Kuka.MovementParameterFieldEnabled=True; ArcTech.WdatVarName=WDAT2; ArcTech.Basic=3.4.3.1264
  ;ENDFOLD
  $BWDSTART = FALSE
  LDAT_ACT = LCPDAT2
  FDAT_ACT = FP4
  BAS(#CP_PARAMS, gArcBasVelDefinition)
  SET_CD_PARAMS (0)
  TRIGGER WHEN PATH = ArcGetPath(#ArcOffBefore, WDAT2) DELAY = 0 DO ArcMainNG(#ArcOffBeforeOffStd, WDAT2, WP4) PRIO = -1
  TRIGGER WHEN PATH = ArcGetPath(#OnTheFlyArcOff, WDAT2) DELAY = 0 DO ArcMainNG(#ArcOffMoveStd, WDAT2, WP4) PRIO = -1
  ArcMainNG(#ArcOffBeforeMoveStd, WDAT2, WP4)
  LIN XP4
  ArcMainNG(#ArcOffAfterMoveStd, WDAT2, WP4)
;ENDFOLD
   $VEL.CP = 0.080
   LIN  {X 0.787, Y -8.829, Z 0.700, A 0.000, B 0.000, C 0.000} C_DIS

;FOLD ARCON WDAT1 LIN P3 Vel=0.5 m/s CPDAT1 Tool[1]:cmttorch Base[1]:vrashatel ;%{PE}
  ;FOLD Parameters ;%{h}
    ;Params IlfProvider=kukaroboter.arctech.arconlin; Kuka.IsGlobalPoint=False; Kuka.PointName=P3; Kuka.BlendingEnabled=False; Kuka.MoveDataName=CPDAT1; Kuka.VelocityPath=0.5; Kuka.CurrentCDSetIndex=0; Kuka.MovementParameterFieldEnabled=True; ArcTech.WdatVarName=WDAT1; ArcTech.Basic=3.4.3.1264
  ;ENDFOLD
  $BWDSTART = FALSE
  LDAT_ACT = LCPDAT1
  FDAT_ACT = FP3
  BAS(#CP_PARAMS, 0.5)
  SET_CD_PARAMS (0)
  TRIGGER WHEN DISTANCE = 1 DELAY = ArcGetDelay(#PreDefinition, WDAT1) DO ArcMainNG(#PreDefinition, WDAT1, WP3) PRIO = -1
  TRIGGER WHEN PATH = ArcGetPath(#OnTheFlyArcOn, WDAT1) DELAY = ArcGetDelay(#GasPreflow, WDAT1) DO ArcMainNG(#GasPreflow, WDAT1, WP3) PRIO = -1
  TRIGGER WHEN PATH = ArcGetPath(#OnTheFlyArcOn, WDAT1) DELAY = 0 DO ArcMainNG(#ArcOnMoveStd, WDAT1, WP3) PRIO = -1
  ArcMainNG(#ArcOnBeforeMoveStd, WDAT1, WP3)
  LIN XP3
  ArcMainNG(#ArcOnAfterMoveStd, WDAT1, WP3)
;ENDFOLD
   $VEL.CP = 0.060
   LIN  {X 8.829, Y -0.787, Z 0.700, A 0.000, B 0.000, C 0.000} C_DIS

;FOLD ARCOFF WDAT2 LIN P4 CPDAT2 Tool[1]:cmttorch Base[1]:vrashatel ;%{PE}
  ;FOLD Parameters ;%{h}
    ;Params IlfProvider=kukaroboter.arctech.arcofflin; Kuka.IsGlobalPoint=False; Kuka.PointName=P4; Kuka.BlendingEnabled=False; Kuka.MoveDataName=CPDAT2; Kuka.VelocityPath=0.01; Kuka.CurrentCDSetIndex=0; Kuka.MovementParameterFieldEnabled=True; ArcTech.WdatVarName=WDAT2; ArcTech.Basic=3.4.3.1264
  ;ENDFOLD
  $BWDSTART = FALSE
  LDAT_ACT = LCPDAT2
  FDAT_ACT = FP4
  BAS(#CP_PARAMS, gArcBasVelDefinition)
  SET_CD_PARAMS (0)
  TRIGGER WHEN PATH = ArcGetPath(#ArcOffBefore, WDAT2) DELAY = 0 DO ArcMainNG(#ArcOffBeforeOffStd, WDAT2, WP4) PRIO = -1
  TRIGGER WHEN PATH = ArcGetPath(#OnTheFlyArcOff, WDAT2) DELAY = 0 DO ArcMainNG(#ArcOffMoveStd, WDAT2, WP4) PRIO = -1
  ArcMainNG(#ArcOffBeforeMoveStd, WDAT2, WP4)
  LIN XP4
  ArcMainNG(#ArcOffAfterMoveStd, WDAT2, WP4)
;ENDFOLD
   $VEL.CP = 0.080
   LIN  {X 8.829, Y -1.352, Z 0.700, A 0.000, B 0.000, C 0.000} C_DIS

;FOLD ARCON WDAT1 LIN P3 Vel=0.5 m/s CPDAT1 Tool[1]:cmttorch Base[1]:vrashatel ;%{PE}
  ;FOLD Parameters ;%{h}
    ;Params IlfProvider=kukaroboter.arctech.arconlin; Kuka.IsGlobalPoint=False; Kuka.PointName=P3; Kuka.BlendingEnabled=False; Kuka.MoveDataName=CPDAT1; Kuka.VelocityPath=0.5; Kuka.CurrentCDSetIndex=0; Kuka.MovementParameterFieldEnabled=True; ArcTech.WdatVarName=WDAT1; ArcTech.Basic=3.4.3.1264
  ;ENDFOLD
  $BWDSTART = FALSE
  LDAT_ACT = LCPDAT1
  FDAT_ACT = FP3
  BAS(#CP_PARAMS, 0.5)
  SET_CD_PARAMS (0)
  TRIGGER WHEN DISTANCE = 1 DELAY = ArcGetDelay(#PreDefinition, WDAT1) DO ArcMainNG(#PreDefinition, WDAT1, WP3) PRIO = -1
  TRIGGER WHEN PATH = ArcGetPath(#OnTheFlyArcOn, WDAT1) DELAY = ArcGetDelay(#GasPreflow, WDAT1) DO ArcMainNG(#GasPreflow, WDAT1, WP3) PRIO = -1
  TRIGGER WHEN PATH = ArcGetPath(#OnTheFlyArcOn, WDAT1) DELAY = 0 DO ArcMainNG(#ArcOnMoveStd, WDAT1, WP3) PRIO = -1
  ArcMainNG(#ArcOnBeforeMoveStd, WDAT1, WP3)
  LIN XP3
  ArcMainNG(#ArcOnAfterMoveStd, WDAT1, WP3)
;ENDFOLD
   $VEL.CP = 0.060
   LIN  {X 1.352, Y -8.829, Z 0.700, A 0.000, B 0.000, C 0.000} C_DIS

;FOLD ARCOFF WDAT2 LIN P4 CPDAT2 Tool[1]:cmttorch Base[1]:vrashatel ;%{PE}
  ;FOLD Parameters ;%{h}
    ;Params IlfProvider=kukaroboter.arctech.arcofflin; Kuka.IsGlobalPoint=False; Kuka.PointName=P4; Kuka.BlendingEnabled=False; Kuka.MoveDataName=CPDAT2; Kuka.VelocityPath=0.01; Kuka.CurrentCDSetIndex=0; Kuka.MovementParameterFieldEnabled=True; ArcTech.WdatVarName=WDAT2; ArcTech.Basic=3.4.3.1264
  ;ENDFOLD
  $BWDSTART = FALSE
  LDAT_ACT = LCPDAT2
  FDAT_ACT = FP4
  BAS(#CP_PARAMS, gArcBasVelDefinition)
  SET_CD_PARAMS (0)
  TRIGGER WHEN PATH = ArcGetPath(#ArcOffBefore, WDAT2) DELAY = 0 DO ArcMainNG(#ArcOffBeforeOffStd, WDAT2, WP4) PRIO = -1
  TRIGGER WHEN PATH = ArcGetPath(#OnTheFlyArcOff, WDAT2) DELAY = 0 DO ArcMainNG(#ArcOffMoveStd, WDAT2, WP4) PRIO = -1
  ArcMainNG(#ArcOffBeforeMoveStd, WDAT2, WP4)
  LIN XP4
  ArcMainNG(#ArcOffAfterMoveStd, WDAT2, WP4)
;ENDFOLD
   $VEL.CP = 0.080
   LIN  {X 1.918, Y -8.829, Z 0.700, A 0.000, B 0.000, C 0.000} C_DIS

;FOLD ARCON WDAT1 LIN P3 Vel=0.5 m/s CPDAT1 Tool[1]:cmttorch Base[1]:vrashatel ;%{PE}
  ;FOLD Parameters ;%{h}
    ;Params IlfProvider=kukaroboter.arctech.arconlin; Kuka.IsGlobalPoint=False; Kuka.PointName=P3; Kuka.BlendingEnabled=False; Kuka.MoveDataName=CPDAT1; Kuka.VelocityPath=0.5; Kuka.CurrentCDSetIndex=0; Kuka.MovementParameterFieldEnabled=True; ArcTech.WdatVarName=WDAT1; ArcTech.Basic=3.4.3.1264
  ;ENDFOLD
  $BWDSTART = FALSE
  LDAT_ACT = LCPDAT1
  FDAT_ACT = FP3
  BAS(#CP_PARAMS, 0.5)
  SET_CD_PARAMS (0)
  TRIGGER WHEN DISTANCE = 1 DELAY = ArcGetDelay(#PreDefinition, WDAT1) DO ArcMainNG(#PreDefinition, WDAT1, WP3) PRIO = -1
  TRIGGER WHEN PATH = ArcGetPath(#OnTheFlyArcOn, WDAT1) DELAY = ArcGetDelay(#GasPreflow, WDAT1) DO ArcMainNG(#GasPreflow, WDAT1, WP3) PRIO = -1
  TRIGGER WHEN PATH = ArcGetPath(#OnTheFlyArcOn, WDAT1) DELAY = 0 DO ArcMainNG(#ArcOnMoveStd, WDAT1, WP3) PRIO = -1
  ArcMainNG(#ArcOnBeforeMoveStd, WDAT1, WP3)
  LIN XP3
  ArcMainNG(#ArcOnAfterMoveStd, WDAT1, WP3)
;ENDFOLD
   $VEL.CP = 0.060
   LIN  {X 8.829, Y -1.918, Z 0.700, A 0.000, B 0.000, C 0.000} C_DIS

;FOLD ARCOFF WDAT2 LIN P4 CPDAT2 Tool[1]:cmttorch Base[1]:vrashatel ;%{PE}
  ;FOLD Parameters ;%{h}
    ;Params IlfProvider=kukaroboter.arctech.arcofflin; Kuka.IsGlobalPoint=False; Kuka.PointName=P4; Kuka.BlendingEnabled=False; Kuka.MoveDataName=CPDAT2; Kuka.VelocityPath=0.01; Kuka.CurrentCDSetIndex=0; Kuka.MovementParameterFieldEnabled=True; ArcTech.WdatVarName=WDAT2; ArcTech.Basic=3.4.3.1264
  ;ENDFOLD
  $BWDSTART = FALSE
  LDAT_ACT = LCPDAT2
  FDAT_ACT = FP4
  BAS(#CP_PARAMS, gArcBasVelDefinition)
  SET_CD_PARAMS (0)
  TRIGGER WHEN PATH = ArcGetPath(#ArcOffBefore, WDAT2) DELAY = 0 DO ArcMainNG(#ArcOffBeforeOffStd, WDAT2, WP4) PRIO = -1
  TRIGGER WHEN PATH = ArcGetPath(#OnTheFlyArcOff, WDAT2) DELAY = 0 DO ArcMainNG(#ArcOffMoveStd, WDAT2, WP4) PRIO = -1
  ArcMainNG(#ArcOffBeforeMoveStd, WDAT2, WP4)
  LIN XP4
  ArcMainNG(#ArcOffAfterMoveStd, WDAT2, WP4)
;ENDFOLD
   $VEL.CP = 0.080
   LIN  {X 8.829, Y -2.484, Z 0.700, A 0.000, B 0.000, C 0.000} C_DIS

;FOLD ARCON WDAT1 LIN P3 Vel=0.5 m/s CPDAT1 Tool[1]:cmttorch Base[1]:vrashatel ;%{PE}
  ;FOLD Parameters ;%{h}
    ;Params IlfProvider=kukaroboter.arctech.arconlin; Kuka.IsGlobalPoint=False; Kuka.PointName=P3; Kuka.BlendingEnabled=False; Kuka.MoveDataName=CPDAT1; Kuka.VelocityPath=0.5; Kuka.CurrentCDSetIndex=0; Kuka.MovementParameterFieldEnabled=True; ArcTech.WdatVarName=WDAT1; ArcTech.Basic=3.4.3.1264
  ;ENDFOLD
  $BWDSTART = FALSE
  LDAT_ACT = LCPDAT1
  FDAT_ACT = FP3
  BAS(#CP_PARAMS, 0.5)
  SET_CD_PARAMS (0)
  TRIGGER WHEN DISTANCE = 1 DELAY = ArcGetDelay(#PreDefinition, WDAT1) DO ArcMainNG(#PreDefinition, WDAT1, WP3) PRIO = -1
  TRIGGER WHEN PATH = ArcGetPath(#OnTheFlyArcOn, WDAT1) DELAY = ArcGetDelay(#GasPreflow, WDAT1) DO ArcMainNG(#GasPreflow, WDAT1, WP3) PRIO = -1
  TRIGGER WHEN PATH = ArcGetPath(#OnTheFlyArcOn, WDAT1) DELAY = 0 DO ArcMainNG(#ArcOnMoveStd, WDAT1, WP3) PRIO = -1
  ArcMainNG(#ArcOnBeforeMoveStd, WDAT1, WP3)
  LIN XP3
  ArcMainNG(#ArcOnAfterMoveStd, WDAT1, WP3)
;ENDFOLD
   $VEL.CP = 0.060
   LIN  {X 2.484, Y -8.829, Z 0.700, A 0.000, B 0.000, C 0.000} C_DIS

;FOLD ARCOFF WDAT2 LIN P4 CPDAT2 Tool[1]:cmttorch Base[1]:vrashatel ;%{PE}
  ;FOLD Parameters ;%{h}
    ;Params IlfProvider=kukaroboter.arctech.arcofflin; Kuka.IsGlobalPoint=False; Kuka.PointName=P4; Kuka.BlendingEnabled=False; Kuka.MoveDataName=CPDAT2; Kuka.VelocityPath=0.01; Kuka.CurrentCDSetIndex=0; Kuka.MovementParameterFieldEnabled=True; ArcTech.WdatVarName=WDAT2; ArcTech.Basic=3.4.3.1264
  ;ENDFOLD
  $BWDSTART = FALSE
  LDAT_ACT = LCPDAT2
  FDAT_ACT = FP4
  BAS(#CP_PARAMS, gArcBasVelDefinition)
  SET_CD_PARAMS (0)
  TRIGGER WHEN PATH = ArcGetPath(#ArcOffBefore, WDAT2) DELAY = 0 DO ArcMainNG(#ArcOffBeforeOffStd, WDAT2, WP4) PRIO = -1
  TRIGGER WHEN PATH = ArcGetPath(#OnTheFlyArcOff, WDAT2) DELAY = 0 DO ArcMainNG(#ArcOffMoveStd, WDAT2, WP4) PRIO = -1
  ArcMainNG(#ArcOffBeforeMoveStd, WDAT2, WP4)
  LIN XP4
  ArcMainNG(#ArcOffAfterMoveStd, WDAT2, WP4)
;ENDFOLD
   $VEL.CP = 0.080
   LIN  {X 3.049, Y -8.829, Z 0.700, A 0.000, B 0.000, C 0.000} C_DIS

;FOLD ARCON WDAT1 LIN P3 Vel=0.5 m/s CPDAT1 Tool[1]:cmttorch Base[1]:vrashatel ;%{PE}
  ;FOLD Parameters ;%{h}
    ;Params IlfProvider=kukaroboter.arctech.arconlin; Kuka.IsGlobalPoint=False; Kuka.PointName=P3; Kuka.BlendingEnabled=False; Kuka.MoveDataName=CPDAT1; Kuka.VelocityPath=0.5; Kuka.CurrentCDSetIndex=0; Kuka.MovementParameterFieldEnabled=True; ArcTech.WdatVarName=WDAT1; ArcTech.Basic=3.4.3.1264
  ;ENDFOLD
  $BWDSTART = FALSE
  LDAT_ACT = LCPDAT1
  FDAT_ACT = FP3
  BAS(#CP_PARAMS, 0.5)
  SET_CD_PARAMS (0)
  TRIGGER WHEN DISTANCE = 1 DELAY = ArcGetDelay(#PreDefinition, WDAT1) DO ArcMainNG(#PreDefinition, WDAT1, WP3) PRIO = -1
  TRIGGER WHEN PATH = ArcGetPath(#OnTheFlyArcOn, WDAT1) DELAY = ArcGetDelay(#GasPreflow, WDAT1) DO ArcMainNG(#GasPreflow, WDAT1, WP3) PRIO = -1
  TRIGGER WHEN PATH = ArcGetPath(#OnTheFlyArcOn, WDAT1) DELAY = 0 DO ArcMainNG(#ArcOnMoveStd, WDAT1, WP3) PRIO = -1
  ArcMainNG(#ArcOnBeforeMoveStd, WDAT1, WP3)
  LIN XP3
  ArcMainNG(#ArcOnAfterMoveStd, WDAT1, WP3)
;ENDFOLD
   $VEL.CP = 0.060
   LIN  {X 8.829, Y -3.049, Z 0.700, A 0.000, B 0.000, C 0.000} C_DIS

;FOLD ARCOFF WDAT2 LIN P4 CPDAT2 Tool[1]:cmttorch Base[1]:vrashatel ;%{PE}
  ;FOLD Parameters ;%{h}
    ;Params IlfProvider=kukaroboter.arctech.arcofflin; Kuka.IsGlobalPoint=False; Kuka.PointName=P4; Kuka.BlendingEnabled=False; Kuka.MoveDataName=CPDAT2; Kuka.VelocityPath=0.01; Kuka.CurrentCDSetIndex=0; Kuka.MovementParameterFieldEnabled=True; ArcTech.WdatVarName=WDAT2; ArcTech.Basic=3.4.3.1264
  ;ENDFOLD
  $BWDSTART = FALSE
  LDAT_ACT = LCPDAT2
  FDAT_ACT = FP4
  BAS(#CP_PARAMS, gArcBasVelDefinition)
  SET_CD_PARAMS (0)
  TRIGGER WHEN PATH = ArcGetPath(#ArcOffBefore, WDAT2) DELAY = 0 DO ArcMainNG(#ArcOffBeforeOffStd, WDAT2, WP4) PRIO = -1
  TRIGGER WHEN PATH = ArcGetPath(#OnTheFlyArcOff, WDAT2) DELAY = 0 DO ArcMainNG(#ArcOffMoveStd, WDAT2, WP4) PRIO = -1
  ArcMainNG(#ArcOffBeforeMoveStd, WDAT2, WP4)
  LIN XP4
  ArcMainNG(#ArcOffAfterMoveStd, WDAT2, WP4)
;ENDFOLD
   $VEL.CP = 0.080
   LIN  {X 8.829, Y -3.615, Z 0.700, A 0.000, B 0.000, C 0.000} C_DIS

;FOLD ARCON WDAT1 LIN P3 Vel=0.5 m/s CPDAT1 Tool[1]:cmttorch Base[1]:vrashatel ;%{PE}
  ;FOLD Parameters ;%{h}
    ;Params IlfProvider=kukaroboter.arctech.arconlin; Kuka.IsGlobalPoint=False; Kuka.PointName=P3; Kuka.BlendingEnabled=False; Kuka.MoveDataName=CPDAT1; Kuka.VelocityPath=0.5; Kuka.CurrentCDSetIndex=0; Kuka.MovementParameterFieldEnabled=True; ArcTech.WdatVarName=WDAT1; ArcTech.Basic=3.4.3.1264
  ;ENDFOLD
  $BWDSTART = FALSE
  LDAT_ACT = LCPDAT1
  FDAT_ACT = FP3
  BAS(#CP_PARAMS, 0.5)
  SET_CD_PARAMS (0)
  TRIGGER WHEN DISTANCE = 1 DELAY = ArcGetDelay(#PreDefinition, WDAT1) DO ArcMainNG(#PreDefinition, WDAT1, WP3) PRIO = -1
  TRIGGER WHEN PATH = ArcGetPath(#OnTheFlyArcOn, WDAT1) DELAY = ArcGetDelay(#GasPreflow, WDAT1) DO ArcMainNG(#GasPreflow, WDAT1, WP3) PRIO = -1
  TRIGGER WHEN PATH = ArcGetPath(#OnTheFlyArcOn, WDAT1) DELAY = 0 DO ArcMainNG(#ArcOnMoveStd, WDAT1, WP3) PRIO = -1
  ArcMainNG(#ArcOnBeforeMoveStd, WDAT1, WP3)
  LIN XP3
  ArcMainNG(#ArcOnAfterMoveStd, WDAT1, WP3)
;ENDFOLD
   $VEL.CP = 0.060
   LIN  {X 3.615, Y -8.829, Z 0.700, A 0.000, B 0.000, C 0.000} C_DIS

;FOLD ARCOFF WDAT2 LIN P4 CPDAT2 Tool[1]:cmttorch Base[1]:vrashatel ;%{PE}
  ;FOLD Parameters ;%{h}
    ;Params IlfProvider=kukaroboter.arctech.arcofflin; Kuka.IsGlobalPoint=False; Kuka.PointName=P4; Kuka.BlendingEnabled=False; Kuka.MoveDataName=CPDAT2; Kuka.VelocityPath=0.01; Kuka.CurrentCDSetIndex=0; Kuka.MovementParameterFieldEnabled=True; ArcTech.WdatVarName=WDAT2; ArcTech.Basic=3.4.3.1264
  ;ENDFOLD
  $BWDSTART = FALSE
  LDAT_ACT = LCPDAT2
  FDAT_ACT = FP4
  BAS(#CP_PARAMS, gArcBasVelDefinition)
  SET_CD_PARAMS (0)
  TRIGGER WHEN PATH = ArcGetPath(#ArcOffBefore, WDAT2) DELAY = 0 DO ArcMainNG(#ArcOffBeforeOffStd, WDAT2, WP4) PRIO = -1
  TRIGGER WHEN PATH = ArcGetPath(#OnTheFlyArcOff, WDAT2) DELAY = 0 DO ArcMainNG(#ArcOffMoveStd, WDAT2, WP4) PRIO = -1
  ArcMainNG(#ArcOffBeforeMoveStd, WDAT2, WP4)
  LIN XP4
  ArcMainNG(#ArcOffAfterMoveStd, WDAT2, WP4)
;ENDFOLD
   $VEL.CP = 0.080
   LIN  {X 4.181, Y -8.829, Z 0.700, A 0.000, B 0.000, C 0.000} C_DIS

;FOLD ARCON WDAT1 LIN P3 Vel=0.5 m/s CPDAT1 Tool[1]:cmttorch Base[1]:vrashatel ;%{PE}
  ;FOLD Parameters ;%{h}
    ;Params IlfProvider=kukaroboter.arctech.arconlin; Kuka.IsGlobalPoint=False; Kuka.PointName=P3; Kuka.BlendingEnabled=False; Kuka.MoveDataName=CPDAT1; Kuka.VelocityPath=0.5; Kuka.CurrentCDSetIndex=0; Kuka.MovementParameterFieldEnabled=True; ArcTech.WdatVarName=WDAT1; ArcTech.Basic=3.4.3.1264
  ;ENDFOLD
  $BWDSTART = FALSE
  LDAT_ACT = LCPDAT1
  FDAT_ACT = FP3
  BAS(#CP_PARAMS, 0.5)
  SET_CD_PARAMS (0)
  TRIGGER WHEN DISTANCE = 1 DELAY = ArcGetDelay(#PreDefinition, WDAT1) DO ArcMainNG(#PreDefinition, WDAT1, WP3) PRIO = -1
  TRIGGER WHEN PATH = ArcGetPath(#OnTheFlyArcOn, WDAT1) DELAY = ArcGetDelay(#GasPreflow, WDAT1) DO ArcMainNG(#GasPreflow, WDAT1, WP3) PRIO = -1
  TRIGGER WHEN PATH = ArcGetPath(#OnTheFlyArcOn, WDAT1) DELAY = 0 DO ArcMainNG(#ArcOnMoveStd, WDAT1, WP3) PRIO = -1
  ArcMainNG(#ArcOnBeforeMoveStd, WDAT1, WP3)
  LIN XP3
  ArcMainNG(#ArcOnAfterMoveStd, WDAT1, WP3)
;ENDFOLD
   $VEL.CP = 0.060
   LIN  {X 8.829, Y -4.181, Z 0.700, A 0.000, B 0.000, C 0.000} C_DIS

;FOLD ARCOFF WDAT2 LIN P4 CPDAT2 Tool[1]:cmttorch Base[1]:vrashatel ;%{PE}
  ;FOLD Parameters ;%{h}
    ;Params IlfProvider=kukaroboter.arctech.arcofflin; Kuka.IsGlobalPoint=False; Kuka.PointName=P4; Kuka.BlendingEnabled=False; Kuka.MoveDataName=CPDAT2; Kuka.VelocityPath=0.01; Kuka.CurrentCDSetIndex=0; Kuka.MovementParameterFieldEnabled=True; ArcTech.WdatVarName=WDAT2; ArcTech.Basic=3.4.3.1264
  ;ENDFOLD
  $BWDSTART = FALSE
  LDAT_ACT = LCPDAT2
  FDAT_ACT = FP4
  BAS(#CP_PARAMS, gArcBasVelDefinition)
  SET_CD_PARAMS (0)
  TRIGGER WHEN PATH = ArcGetPath(#ArcOffBefore, WDAT2) DELAY = 0 DO ArcMainNG(#ArcOffBeforeOffStd, WDAT2, WP4) PRIO = -1
  TRIGGER WHEN PATH = ArcGetPath(#OnTheFlyArcOff, WDAT2) DELAY = 0 DO ArcMainNG(#ArcOffMoveStd, WDAT2, WP4) PRIO = -1
  ArcMainNG(#ArcOffBeforeMoveStd, WDAT2, WP4)
  LIN XP4
  ArcMainNG(#ArcOffAfterMoveStd, WDAT2, WP4)
;ENDFOLD
   $VEL.CP = 0.080
   LIN  {X 8.829, Y -4.746, Z 0.700, A 0.000, B 0.000, C 0.000} C_DIS

;FOLD ARCON WDAT1 LIN P3 Vel=0.5 m/s CPDAT1 Tool[1]:cmttorch Base[1]:vrashatel ;%{PE}
  ;FOLD Parameters ;%{h}
    ;Params IlfProvider=kukaroboter.arctech.arconlin; Kuka.IsGlobalPoint=False; Kuka.PointName=P3; Kuka.BlendingEnabled=False; Kuka.MoveDataName=CPDAT1; Kuka.VelocityPath=0.5; Kuka.CurrentCDSetIndex=0; Kuka.MovementParameterFieldEnabled=True; ArcTech.WdatVarName=WDAT1; ArcTech.Basic=3.4.3.1264
  ;ENDFOLD
  $BWDSTART = FALSE
  LDAT_ACT = LCPDAT1
  FDAT_ACT = FP3
  BAS(#CP_PARAMS, 0.5)
  SET_CD_PARAMS (0)
  TRIGGER WHEN DISTANCE = 1 DELAY = ArcGetDelay(#PreDefinition, WDAT1) DO ArcMainNG(#PreDefinition, WDAT1, WP3) PRIO = -1
  TRIGGER WHEN PATH = ArcGetPath(#OnTheFlyArcOn, WDAT1) DELAY = ArcGetDelay(#GasPreflow, WDAT1) DO ArcMainNG(#GasPreflow, WDAT1, WP3) PRIO = -1
  TRIGGER WHEN PATH = ArcGetPath(#OnTheFlyArcOn, WDAT1) DELAY = 0 DO ArcMainNG(#ArcOnMoveStd, WDAT1, WP3) PRIO = -1
  ArcMainNG(#ArcOnBeforeMoveStd, WDAT1, WP3)
  LIN XP3
  ArcMainNG(#ArcOnAfterMoveStd, WDAT1, WP3)
;ENDFOLD
   $VEL.CP = 0.060
   LIN  {X 4.746, Y -8.829, Z 0.700, A 0.000, B 0.000, C 0.000} C_DIS

;FOLD ARCOFF WDAT2 LIN P4 CPDAT2 Tool[1]:cmttorch Base[1]:vrashatel ;%{PE}
  ;FOLD Parameters ;%{h}
    ;Params IlfProvider=kukaroboter.arctech.arcofflin; Kuka.IsGlobalPoint=False; Kuka.PointName=P4; Kuka.BlendingEnabled=False; Kuka.MoveDataName=CPDAT2; Kuka.VelocityPath=0.01; Kuka.CurrentCDSetIndex=0; Kuka.MovementParameterFieldEnabled=True; ArcTech.WdatVarName=WDAT2; ArcTech.Basic=3.4.3.1264
  ;ENDFOLD
  $BWDSTART = FALSE
  LDAT_ACT = LCPDAT2
  FDAT_ACT = FP4
  BAS(#CP_PARAMS, gArcBasVelDefinition)
  SET_CD_PARAMS (0)
  TRIGGER WHEN PATH = ArcGetPath(#ArcOffBefore, WDAT2) DELAY = 0 DO ArcMainNG(#ArcOffBeforeOffStd, WDAT2, WP4) PRIO = -1
  TRIGGER WHEN PATH = ArcGetPath(#OnTheFlyArcOff, WDAT2) DELAY = 0 DO ArcMainNG(#ArcOffMoveStd, WDAT2, WP4) PRIO = -1
  ArcMainNG(#ArcOffBeforeMoveStd, WDAT2, WP4)
  LIN XP4
  ArcMainNG(#ArcOffAfterMoveStd, WDAT2, WP4)
;ENDFOLD
   $VEL.CP = 0.080
   LIN  {X 5.312, Y -8.829, Z 0.700, A 0.000, B 0.000, C 0.000} C_DIS

;FOLD ARCON WDAT1 LIN P3 Vel=0.5 m/s CPDAT1 Tool[1]:cmttorch Base[1]:vrashatel ;%{PE}
  ;FOLD Parameters ;%{h}
    ;Params IlfProvider=kukaroboter.arctech.arconlin; Kuka.IsGlobalPoint=False; Kuka.PointName=P3; Kuka.BlendingEnabled=False; Kuka.MoveDataName=CPDAT1; Kuka.VelocityPath=0.5; Kuka.CurrentCDSetIndex=0; Kuka.MovementParameterFieldEnabled=True; ArcTech.WdatVarName=WDAT1; ArcTech.Basic=3.4.3.1264
  ;ENDFOLD
  $BWDSTART = FALSE
  LDAT_ACT = LCPDAT1
  FDAT_ACT = FP3
  BAS(#CP_PARAMS, 0.5)
  SET_CD_PARAMS (0)
  TRIGGER WHEN DISTANCE = 1 DELAY = ArcGetDelay(#PreDefinition, WDAT1) DO ArcMainNG(#PreDefinition, WDAT1, WP3) PRIO = -1
  TRIGGER WHEN PATH = ArcGetPath(#OnTheFlyArcOn, WDAT1) DELAY = ArcGetDelay(#GasPreflow, WDAT1) DO ArcMainNG(#GasPreflow, WDAT1, WP3) PRIO = -1
  TRIGGER WHEN PATH = ArcGetPath(#OnTheFlyArcOn, WDAT1) DELAY = 0 DO ArcMainNG(#ArcOnMoveStd, WDAT1, WP3) PRIO = -1
  ArcMainNG(#ArcOnBeforeMoveStd, WDAT1, WP3)
  LIN XP3
  ArcMainNG(#ArcOnAfterMoveStd, WDAT1, WP3)
;ENDFOLD
   $VEL.CP = 0.060
   LIN  {X 8.829, Y -5.312, Z 0.700, A 0.000, B 0.000, C 0.000} C_DIS

;FOLD ARCOFF WDAT2 LIN P4 CPDAT2 Tool[1]:cmttorch Base[1]:vrashatel ;%{PE}
  ;FOLD Parameters ;%{h}
    ;Params IlfProvider=kukaroboter.arctech.arcofflin; Kuka.IsGlobalPoint=False; Kuka.PointName=P4; Kuka.BlendingEnabled=False; Kuka.MoveDataName=CPDAT2; Kuka.VelocityPath=0.01; Kuka.CurrentCDSetIndex=0; Kuka.MovementParameterFieldEnabled=True; ArcTech.WdatVarName=WDAT2; ArcTech.Basic=3.4.3.1264
  ;ENDFOLD
  $BWDSTART = FALSE
  LDAT_ACT = LCPDAT2
  FDAT_ACT = FP4
  BAS(#CP_PARAMS, gArcBasVelDefinition)
  SET_CD_PARAMS (0)
  TRIGGER WHEN PATH = ArcGetPath(#ArcOffBefore, WDAT2) DELAY = 0 DO ArcMainNG(#ArcOffBeforeOffStd, WDAT2, WP4) PRIO = -1
  TRIGGER WHEN PATH = ArcGetPath(#OnTheFlyArcOff, WDAT2) DELAY = 0 DO ArcMainNG(#ArcOffMoveStd, WDAT2, WP4) PRIO = -1
  ArcMainNG(#ArcOffBeforeMoveStd, WDAT2, WP4)
  LIN XP4
  ArcMainNG(#ArcOffAfterMoveStd, WDAT2, WP4)
;ENDFOLD
   $VEL.CP = 0.080
   LIN  {X 8.829, Y -5.878, Z 0.700, A 0.000, B 0.000, C 0.000} C_DIS

;FOLD ARCON WDAT1 LIN P3 Vel=0.5 m/s CPDAT1 Tool[1]:cmttorch Base[1]:vrashatel ;%{PE}
  ;FOLD Parameters ;%{h}
    ;Params IlfProvider=kukaroboter.arctech.arconlin; Kuka.IsGlobalPoint=False; Kuka.PointName=P3; Kuka.BlendingEnabled=False; Kuka.MoveDataName=CPDAT1; Kuka.VelocityPath=0.5; Kuka.CurrentCDSetIndex=0; Kuka.MovementParameterFieldEnabled=True; ArcTech.WdatVarName=WDAT1; ArcTech.Basic=3.4.3.1264
  ;ENDFOLD
  $BWDSTART = FALSE
  LDAT_ACT = LCPDAT1
  FDAT_ACT = FP3
  BAS(#CP_PARAMS, 0.5)
  SET_CD_PARAMS (0)
  TRIGGER WHEN DISTANCE = 1 DELAY = ArcGetDelay(#PreDefinition, WDAT1) DO ArcMainNG(#PreDefinition, WDAT1, WP3) PRIO = -1
  TRIGGER WHEN PATH = ArcGetPath(#OnTheFlyArcOn, WDAT1) DELAY = ArcGetDelay(#GasPreflow, WDAT1) DO ArcMainNG(#GasPreflow, WDAT1, WP3) PRIO = -1
  TRIGGER WHEN PATH = ArcGetPath(#OnTheFlyArcOn, WDAT1) DELAY = 0 DO ArcMainNG(#ArcOnMoveStd, WDAT1, WP3) PRIO = -1
  ArcMainNG(#ArcOnBeforeMoveStd, WDAT1, WP3)
  LIN XP3
  ArcMainNG(#ArcOnAfterMoveStd, WDAT1, WP3)
;ENDFOLD
   $VEL.CP = 0.060
   LIN  {X 5.878, Y -8.829, Z 0.700, A 0.000, B 0.000, C 0.000} C_DIS

;FOLD ARCOFF WDAT2 LIN P4 CPDAT2 Tool[1]:cmttorch Base[1]:vrashatel ;%{PE}
  ;FOLD Parameters ;%{h}
    ;Params IlfProvider=kukaroboter.arctech.arcofflin; Kuka.IsGlobalPoint=False; Kuka.PointName=P4; Kuka.BlendingEnabled=False; Kuka.MoveDataName=CPDAT2; Kuka.VelocityPath=0.01; Kuka.CurrentCDSetIndex=0; Kuka.MovementParameterFieldEnabled=True; ArcTech.WdatVarName=WDAT2; ArcTech.Basic=3.4.3.1264
  ;ENDFOLD
  $BWDSTART = FALSE
  LDAT_ACT = LCPDAT2
  FDAT_ACT = FP4
  BAS(#CP_PARAMS, gArcBasVelDefinition)
  SET_CD_PARAMS (0)
  TRIGGER WHEN PATH = ArcGetPath(#ArcOffBefore, WDAT2) DELAY = 0 DO ArcMainNG(#ArcOffBeforeOffStd, WDAT2, WP4) PRIO = -1
  TRIGGER WHEN PATH = ArcGetPath(#OnTheFlyArcOff, WDAT2) DELAY = 0 DO ArcMainNG(#ArcOffMoveStd, WDAT2, WP4) PRIO = -1
  ArcMainNG(#ArcOffBeforeMoveStd, WDAT2, WP4)
  LIN XP4
  ArcMainNG(#ArcOffAfterMoveStd, WDAT2, WP4)
;ENDFOLD
   $VEL.CP = 0.080
   LIN  {X 6.443, Y -8.829, Z 0.700, A 0.000, B 0.000, C 0.000} C_DIS

;FOLD ARCON WDAT1 LIN P3 Vel=0.5 m/s CPDAT1 Tool[1]:cmttorch Base[1]:vrashatel ;%{PE}
  ;FOLD Parameters ;%{h}
    ;Params IlfProvider=kukaroboter.arctech.arconlin; Kuka.IsGlobalPoint=False; Kuka.PointName=P3; Kuka.BlendingEnabled=False; Kuka.MoveDataName=CPDAT1; Kuka.VelocityPath=0.5; Kuka.CurrentCDSetIndex=0; Kuka.MovementParameterFieldEnabled=True; ArcTech.WdatVarName=WDAT1; ArcTech.Basic=3.4.3.1264
  ;ENDFOLD
  $BWDSTART = FALSE
  LDAT_ACT = LCPDAT1
  FDAT_ACT = FP3
  BAS(#CP_PARAMS, 0.5)
  SET_CD_PARAMS (0)
  TRIGGER WHEN DISTANCE = 1 DELAY = ArcGetDelay(#PreDefinition, WDAT1) DO ArcMainNG(#PreDefinition, WDAT1, WP3) PRIO = -1
  TRIGGER WHEN PATH = ArcGetPath(#OnTheFlyArcOn, WDAT1) DELAY = ArcGetDelay(#GasPreflow, WDAT1) DO ArcMainNG(#GasPreflow, WDAT1, WP3) PRIO = -1
  TRIGGER WHEN PATH = ArcGetPath(#OnTheFlyArcOn, WDAT1) DELAY = 0 DO ArcMainNG(#ArcOnMoveStd, WDAT1, WP3) PRIO = -1
  ArcMainNG(#ArcOnBeforeMoveStd, WDAT1, WP3)
  LIN XP3
  ArcMainNG(#ArcOnAfterMoveStd, WDAT1, WP3)
;ENDFOLD
   $VEL.CP = 0.060
   LIN  {X 8.829, Y -6.443, Z 0.700, A 0.000, B 0.000, C 0.000} C_DIS

;FOLD ARCOFF WDAT2 LIN P4 CPDAT2 Tool[1]:cmttorch Base[1]:vrashatel ;%{PE}
  ;FOLD Parameters ;%{h}
    ;Params IlfProvider=kukaroboter.arctech.arcofflin; Kuka.IsGlobalPoint=False; Kuka.PointName=P4; Kuka.BlendingEnabled=False; Kuka.MoveDataName=CPDAT2; Kuka.VelocityPath=0.01; Kuka.CurrentCDSetIndex=0; Kuka.MovementParameterFieldEnabled=True; ArcTech.WdatVarName=WDAT2; ArcTech.Basic=3.4.3.1264
  ;ENDFOLD
  $BWDSTART = FALSE
  LDAT_ACT = LCPDAT2
  FDAT_ACT = FP4
  BAS(#CP_PARAMS, gArcBasVelDefinition)
  SET_CD_PARAMS (0)
  TRIGGER WHEN PATH = ArcGetPath(#ArcOffBefore, WDAT2) DELAY = 0 DO ArcMainNG(#ArcOffBeforeOffStd, WDAT2, WP4) PRIO = -1
  TRIGGER WHEN PATH = ArcGetPath(#OnTheFlyArcOff, WDAT2) DELAY = 0 DO ArcMainNG(#ArcOffMoveStd, WDAT2, WP4) PRIO = -1
  ArcMainNG(#ArcOffBeforeMoveStd, WDAT2, WP4)
  LIN XP4
  ArcMainNG(#ArcOffAfterMoveStd, WDAT2, WP4)
;ENDFOLD
   $VEL.CP = 0.080
   LIN  {X 8.829, Y -7.009, Z 0.700, A 0.000, B 0.000, C 0.000} C_DIS

;FOLD ARCON WDAT1 LIN P3 Vel=0.5 m/s CPDAT1 Tool[1]:cmttorch Base[1]:vrashatel ;%{PE}
  ;FOLD Parameters ;%{h}
    ;Params IlfProvider=kukaroboter.arctech.arconlin; Kuka.IsGlobalPoint=False; Kuka.PointName=P3; Kuka.BlendingEnabled=False; Kuka.MoveDataName=CPDAT1; Kuka.VelocityPath=0.5; Kuka.CurrentCDSetIndex=0; Kuka.MovementParameterFieldEnabled=True; ArcTech.WdatVarName=WDAT1; ArcTech.Basic=3.4.3.1264
  ;ENDFOLD
  $BWDSTART = FALSE
  LDAT_ACT = LCPDAT1
  FDAT_ACT = FP3
  BAS(#CP_PARAMS, 0.5)
  SET_CD_PARAMS (0)
  TRIGGER WHEN DISTANCE = 1 DELAY = ArcGetDelay(#PreDefinition, WDAT1) DO ArcMainNG(#PreDefinition, WDAT1, WP3) PRIO = -1
  TRIGGER WHEN PATH = ArcGetPath(#OnTheFlyArcOn, WDAT1) DELAY = ArcGetDelay(#GasPreflow, WDAT1) DO ArcMainNG(#GasPreflow, WDAT1, WP3) PRIO = -1
  TRIGGER WHEN PATH = ArcGetPath(#OnTheFlyArcOn, WDAT1) DELAY = 0 DO ArcMainNG(#ArcOnMoveStd, WDAT1, WP3) PRIO = -1
  ArcMainNG(#ArcOnBeforeMoveStd, WDAT1, WP3)
  LIN XP3
  ArcMainNG(#ArcOnAfterMoveStd, WDAT1, WP3)
;ENDFOLD
   $VEL.CP = 0.060
   LIN  {X 7.009, Y -8.829, Z 0.700, A 0.000, B 0.000, C 0.000} C_DIS

;FOLD ARCOFF WDAT2 LIN P4 CPDAT2 Tool[1]:cmttorch Base[1]:vrashatel ;%{PE}
  ;FOLD Parameters ;%{h}
    ;Params IlfProvider=kukaroboter.arctech.arcofflin; Kuka.IsGlobalPoint=False; Kuka.PointName=P4; Kuka.BlendingEnabled=False; Kuka.MoveDataName=CPDAT2; Kuka.VelocityPath=0.01; Kuka.CurrentCDSetIndex=0; Kuka.MovementParameterFieldEnabled=True; ArcTech.WdatVarName=WDAT2; ArcTech.Basic=3.4.3.1264
  ;ENDFOLD
  $BWDSTART = FALSE
  LDAT_ACT = LCPDAT2
  FDAT_ACT = FP4
  BAS(#CP_PARAMS, gArcBasVelDefinition)
  SET_CD_PARAMS (0)
  TRIGGER WHEN PATH = ArcGetPath(#ArcOffBefore, WDAT2) DELAY = 0 DO ArcMainNG(#ArcOffBeforeOffStd, WDAT2, WP4) PRIO = -1
  TRIGGER WHEN PATH = ArcGetPath(#OnTheFlyArcOff, WDAT2) DELAY = 0 DO ArcMainNG(#ArcOffMoveStd, WDAT2, WP4) PRIO = -1
  ArcMainNG(#ArcOffBeforeMoveStd, WDAT2, WP4)
  LIN XP4
  ArcMainNG(#ArcOffAfterMoveStd, WDAT2, WP4)
;ENDFOLD
   $VEL.CP = 0.080
   LIN  {X 7.575, Y -8.829, Z 0.700, A 0.000, B 0.000, C 0.000} C_DIS

;FOLD ARCON WDAT1 LIN P3 Vel=0.5 m/s CPDAT1 Tool[1]:cmttorch Base[1]:vrashatel ;%{PE}
  ;FOLD Parameters ;%{h}
    ;Params IlfProvider=kukaroboter.arctech.arconlin; Kuka.IsGlobalPoint=False; Kuka.PointName=P3; Kuka.BlendingEnabled=False; Kuka.MoveDataName=CPDAT1; Kuka.VelocityPath=0.5; Kuka.CurrentCDSetIndex=0; Kuka.MovementParameterFieldEnabled=True; ArcTech.WdatVarName=WDAT1; ArcTech.Basic=3.4.3.1264
  ;ENDFOLD
  $BWDSTART = FALSE
  LDAT_ACT = LCPDAT1
  FDAT_ACT = FP3
  BAS(#CP_PARAMS, 0.5)
  SET_CD_PARAMS (0)
  TRIGGER WHEN DISTANCE = 1 DELAY = ArcGetDelay(#PreDefinition, WDAT1) DO ArcMainNG(#PreDefinition, WDAT1, WP3) PRIO = -1
  TRIGGER WHEN PATH = ArcGetPath(#OnTheFlyArcOn, WDAT1) DELAY = ArcGetDelay(#GasPreflow, WDAT1) DO ArcMainNG(#GasPreflow, WDAT1, WP3) PRIO = -1
  TRIGGER WHEN PATH = ArcGetPath(#OnTheFlyArcOn, WDAT1) DELAY = 0 DO ArcMainNG(#ArcOnMoveStd, WDAT1, WP3) PRIO = -1
  ArcMainNG(#ArcOnBeforeMoveStd, WDAT1, WP3)
  LIN XP3
  ArcMainNG(#ArcOnAfterMoveStd, WDAT1, WP3)
;ENDFOLD
   $VEL.CP = 0.060
   LIN  {X 8.829, Y -7.575, Z 0.700, A 0.000, B 0.000, C 0.000} C_DIS

;FOLD ARCOFF WDAT2 LIN P4 CPDAT2 Tool[1]:cmttorch Base[1]:vrashatel ;%{PE}
  ;FOLD Parameters ;%{h}
    ;Params IlfProvider=kukaroboter.arctech.arcofflin; Kuka.IsGlobalPoint=False; Kuka.PointName=P4; Kuka.BlendingEnabled=False; Kuka.MoveDataName=CPDAT2; Kuka.VelocityPath=0.01; Kuka.CurrentCDSetIndex=0; Kuka.MovementParameterFieldEnabled=True; ArcTech.WdatVarName=WDAT2; ArcTech.Basic=3.4.3.1264
  ;ENDFOLD
  $BWDSTART = FALSE
  LDAT_ACT = LCPDAT2
  FDAT_ACT = FP4
  BAS(#CP_PARAMS, gArcBasVelDefinition)
  SET_CD_PARAMS (0)
  TRIGGER WHEN PATH = ArcGetPath(#ArcOffBefore, WDAT2) DELAY = 0 DO ArcMainNG(#ArcOffBeforeOffStd, WDAT2, WP4) PRIO = -1
  TRIGGER WHEN PATH = ArcGetPath(#OnTheFlyArcOff, WDAT2) DELAY = 0 DO ArcMainNG(#ArcOffMoveStd, WDAT2, WP4) PRIO = -1
  ArcMainNG(#ArcOffBeforeMoveStd, WDAT2, WP4)
  LIN XP4
  ArcMainNG(#ArcOffAfterMoveStd, WDAT2, WP4)
;ENDFOLD
   $VEL.CP = 0.080
   LIN  {X 8.829, Y -8.140, Z 0.700, A 0.000, B 0.000, C 0.000} C_DIS

;FOLD ARCON WDAT1 LIN P3 Vel=0.5 m/s CPDAT1 Tool[1]:cmttorch Base[1]:vrashatel ;%{PE}
  ;FOLD Parameters ;%{h}
    ;Params IlfProvider=kukaroboter.arctech.arconlin; Kuka.IsGlobalPoint=False; Kuka.PointName=P3; Kuka.BlendingEnabled=False; Kuka.MoveDataName=CPDAT1; Kuka.VelocityPath=0.5; Kuka.CurrentCDSetIndex=0; Kuka.MovementParameterFieldEnabled=True; ArcTech.WdatVarName=WDAT1; ArcTech.Basic=3.4.3.1264
  ;ENDFOLD
  $BWDSTART = FALSE
  LDAT_ACT = LCPDAT1
  FDAT_ACT = FP3
  BAS(#CP_PARAMS, 0.5)
  SET_CD_PARAMS (0)
  TRIGGER WHEN DISTANCE = 1 DELAY = ArcGetDelay(#PreDefinition, WDAT1) DO ArcMainNG(#PreDefinition, WDAT1, WP3) PRIO = -1
  TRIGGER WHEN PATH = ArcGetPath(#OnTheFlyArcOn, WDAT1) DELAY = ArcGetDelay(#GasPreflow, WDAT1) DO ArcMainNG(#GasPreflow, WDAT1, WP3) PRIO = -1
  TRIGGER WHEN PATH = ArcGetPath(#OnTheFlyArcOn, WDAT1) DELAY = 0 DO ArcMainNG(#ArcOnMoveStd, WDAT1, WP3) PRIO = -1
  ArcMainNG(#ArcOnBeforeMoveStd, WDAT1, WP3)
  LIN XP3
  ArcMainNG(#ArcOnAfterMoveStd, WDAT1, WP3)
;ENDFOLD
   $VEL.CP = 0.060
   LIN  {X 8.140, Y -8.829, Z 0.700, A 0.000, B 0.000, C 0.000} C_DIS

;FOLD ARCOFF WDAT2 LIN P4 CPDAT2 Tool[1]:cmttorch Base[1]:vrashatel ;%{PE}
  ;FOLD Parameters ;%{h}
    ;Params IlfProvider=kukaroboter.arctech.arcofflin; Kuka.IsGlobalPoint=False; Kuka.PointName=P4; Kuka.BlendingEnabled=False; Kuka.MoveDataName=CPDAT2; Kuka.VelocityPath=0.01; Kuka.CurrentCDSetIndex=0; Kuka.MovementParameterFieldEnabled=True; ArcTech.WdatVarName=WDAT2; ArcTech.Basic=3.4.3.1264
  ;ENDFOLD
  $BWDSTART = FALSE
  LDAT_ACT = LCPDAT2
  FDAT_ACT = FP4
  BAS(#CP_PARAMS, gArcBasVelDefinition)
  SET_CD_PARAMS (0)
  TRIGGER WHEN PATH = ArcGetPath(#ArcOffBefore, WDAT2) DELAY = 0 DO ArcMainNG(#ArcOffBeforeOffStd, WDAT2, WP4) PRIO = -1
  TRIGGER WHEN PATH = ArcGetPath(#OnTheFlyArcOff, WDAT2) DELAY = 0 DO ArcMainNG(#ArcOffMoveStd, WDAT2, WP4) PRIO = -1
  ArcMainNG(#ArcOffBeforeMoveStd, WDAT2, WP4)
  LIN XP4
  ArcMainNG(#ArcOffAfterMoveStd, WDAT2, WP4)
;ENDFOLD
   $VEL.CP = 0.080
   LIN  {X 8.706, Y -8.829, Z 0.700, A 0.000, B 0.000, C 0.000} C_DIS

;FOLD ARCON WDAT1 LIN P3 Vel=0.5 m/s CPDAT1 Tool[1]:cmttorch Base[1]:vrashatel ;%{PE}
  ;FOLD Parameters ;%{h}
    ;Params IlfProvider=kukaroboter.arctech.arconlin; Kuka.IsGlobalPoint=False; Kuka.PointName=P3; Kuka.BlendingEnabled=False; Kuka.MoveDataName=CPDAT1; Kuka.VelocityPath=0.5; Kuka.CurrentCDSetIndex=0; Kuka.MovementParameterFieldEnabled=True; ArcTech.WdatVarName=WDAT1; ArcTech.Basic=3.4.3.1264
  ;ENDFOLD
  $BWDSTART = FALSE
  LDAT_ACT = LCPDAT1
  FDAT_ACT = FP3
  BAS(#CP_PARAMS, 0.5)
  SET_CD_PARAMS (0)
  TRIGGER WHEN DISTANCE = 1 DELAY = ArcGetDelay(#PreDefinition, WDAT1) DO ArcMainNG(#PreDefinition, WDAT1, WP3) PRIO = -1
  TRIGGER WHEN PATH = ArcGetPath(#OnTheFlyArcOn, WDAT1) DELAY = ArcGetDelay(#GasPreflow, WDAT1) DO ArcMainNG(#GasPreflow, WDAT1, WP3) PRIO = -1
  TRIGGER WHEN PATH = ArcGetPath(#OnTheFlyArcOn, WDAT1) DELAY = 0 DO ArcMainNG(#ArcOnMoveStd, WDAT1, WP3) PRIO = -1
  ArcMainNG(#ArcOnBeforeMoveStd, WDAT1, WP3)
  LIN XP3
  ArcMainNG(#ArcOnAfterMoveStd, WDAT1, WP3)
;ENDFOLD
   $VEL.CP = 0.060
   LIN  {X 8.829, Y -8.706, Z 0.700, A 0.000, B 0.000, C 0.000} C_DIS

;FOLD ARCOFF WDAT2 LIN P4 CPDAT2 Tool[1]:cmttorch Base[1]:vrashatel ;%{PE}
  ;FOLD Parameters ;%{h}
    ;Params IlfProvider=kukaroboter.arctech.arcofflin; Kuka.IsGlobalPoint=False; Kuka.PointName=P4; Kuka.BlendingEnabled=False; Kuka.MoveDataName=CPDAT2; Kuka.VelocityPath=0.01; Kuka.CurrentCDSetIndex=0; Kuka.MovementParameterFieldEnabled=True; ArcTech.WdatVarName=WDAT2; ArcTech.Basic=3.4.3.1264
  ;ENDFOLD
  $BWDSTART = FALSE
  LDAT_ACT = LCPDAT2
  FDAT_ACT = FP4
  BAS(#CP_PARAMS, gArcBasVelDefinition)
  SET_CD_PARAMS (0)
  TRIGGER WHEN PATH = ArcGetPath(#ArcOffBefore, WDAT2) DELAY = 0 DO ArcMainNG(#ArcOffBeforeOffStd, WDAT2, WP4) PRIO = -1
  TRIGGER WHEN PATH = ArcGetPath(#OnTheFlyArcOff, WDAT2) DELAY = 0 DO ArcMainNG(#ArcOffMoveStd, WDAT2, WP4) PRIO = -1
  ArcMainNG(#ArcOffBeforeMoveStd, WDAT2, WP4)
  LIN XP4
  ArcMainNG(#ArcOffAfterMoveStd, WDAT2, WP4)
;ENDFOLD
   $VEL.CP = 0.080
   LIN  {X 9.200, Y -8.706, Z 0.700, A 0.000, B 0.000, C 0.000} C_DIS
   $VEL.CP = 0.010
   LIN  {X 9.200, Y -8.706, Z 0.900, A 0.000, B 0.000, C 0.000} C_DIS
   $VEL.CP = 0.080
   LIN  {X 9.290, Y -8.706, Z 0.900, A 0.000, B 0.000, C 0.000} C_DIS
   $VEL.CP = 0.080
   LIN  {X 9.218, Y 9.218, Z 0.900, A 0.000, B 0.000, C 0.000} C_DIS
   $VEL.CP = 0.080
   LIN  {X -9.530, Y 9.530, Z 0.900, A 0.000, B 0.000, C 0.000} C_DIS
   $VEL.CP = 0.080
   LIN  {X -9.800, Y 9.800, Z 0.900, A 0.000, B 0.000, C 0.000} C_DIS

;FOLD ARCON WDAT1 LIN P3 Vel=0.5 m/s CPDAT1 Tool[1]:cmttorch Base[1]:vrashatel ;%{PE}
  ;FOLD Parameters ;%{h}
    ;Params IlfProvider=kukaroboter.arctech.arconlin; Kuka.IsGlobalPoint=False; Kuka.PointName=P3; Kuka.BlendingEnabled=False; Kuka.MoveDataName=CPDAT1; Kuka.VelocityPath=0.5; Kuka.CurrentCDSetIndex=0; Kuka.MovementParameterFieldEnabled=True; ArcTech.WdatVarName=WDAT1; ArcTech.Basic=3.4.3.1264
  ;ENDFOLD
  $BWDSTART = FALSE
  LDAT_ACT = LCPDAT1
  FDAT_ACT = FP3
  BAS(#CP_PARAMS, 0.5)
  SET_CD_PARAMS (0)
  TRIGGER WHEN DISTANCE = 1 DELAY = ArcGetDelay(#PreDefinition, WDAT1) DO ArcMainNG(#PreDefinition, WDAT1, WP3) PRIO = -1
  TRIGGER WHEN PATH = ArcGetPath(#OnTheFlyArcOn, WDAT1) DELAY = ArcGetDelay(#GasPreflow, WDAT1) DO ArcMainNG(#GasPreflow, WDAT1, WP3) PRIO = -1
  TRIGGER WHEN PATH = ArcGetPath(#OnTheFlyArcOn, WDAT1) DELAY = 0 DO ArcMainNG(#ArcOnMoveStd, WDAT1, WP3) PRIO = -1
  ArcMainNG(#ArcOnBeforeMoveStd, WDAT1, WP3)
  LIN XP3
  ArcMainNG(#ArcOnAfterMoveStd, WDAT1, WP3)
;ENDFOLD
   $VEL.CP = 0.025
   LIN  {X -9.800, Y 9.800, Z 0.900, A 0.000, B 0.000, C 0.000} C_DIS
   $VEL.CP = 0.060
   LIN  {X -9.800, Y -9.800, Z 0.900, A 0.000, B 0.000, C 0.000} C_DIS
   $VEL.CP = 0.060
   LIN  {X 9.800, Y -9.800, Z 0.900, A 0.000, B 0.000, C 0.000} C_DIS
   $VEL.CP = 0.060
   LIN  {X 9.800, Y 9.800, Z 0.900, A 0.000, B 0.000, C 0.000} C_DIS
   $VEL.CP = 0.060
   LIN  {X -9.800, Y 9.800, Z 0.900, A 0.000, B 0.000, C 0.000} C_DIS

;FOLD ARCOFF WDAT2 LIN P4 CPDAT2 Tool[1]:cmttorch Base[1]:vrashatel ;%{PE}
  ;FOLD Parameters ;%{h}
    ;Params IlfProvider=kukaroboter.arctech.arcofflin; Kuka.IsGlobalPoint=False; Kuka.PointName=P4; Kuka.BlendingEnabled=False; Kuka.MoveDataName=CPDAT2; Kuka.VelocityPath=0.01; Kuka.CurrentCDSetIndex=0; Kuka.MovementParameterFieldEnabled=True; ArcTech.WdatVarName=WDAT2; ArcTech.Basic=3.4.3.1264
  ;ENDFOLD
  $BWDSTART = FALSE
  LDAT_ACT = LCPDAT2
  FDAT_ACT = FP4
  BAS(#CP_PARAMS, gArcBasVelDefinition)
  SET_CD_PARAMS (0)
  TRIGGER WHEN PATH = ArcGetPath(#ArcOffBefore, WDAT2) DELAY = 0 DO ArcMainNG(#ArcOffBeforeOffStd, WDAT2, WP4) PRIO = -1
  TRIGGER WHEN PATH = ArcGetPath(#OnTheFlyArcOff, WDAT2) DELAY = 0 DO ArcMainNG(#ArcOffMoveStd, WDAT2, WP4) PRIO = -1
  ArcMainNG(#ArcOffBeforeMoveStd, WDAT2, WP4)
  LIN XP4
  ArcMainNG(#ArcOffAfterMoveStd, WDAT2, WP4)
;ENDFOLD
   $VEL.CP = 0.080
   LIN  {X -9.800, Y 9.600, Z 0.900, A 0.000, B 0.000, C 0.000} C_DIS
   $VEL.CP = 0.080
   LIN  {X -9.360, Y 9.360, Z 0.900, A 0.000, B 0.000, C 0.000} C_DIS
   $VEL.CP = 0.080
   LIN  {X -9.400, Y 9.400, Z 0.900, A 0.000, B 0.000, C 0.000} C_DIS

;FOLD ARCON WDAT1 LIN P3 Vel=0.5 m/s CPDAT1 Tool[1]:cmttorch Base[1]:vrashatel ;%{PE}
  ;FOLD Parameters ;%{h}
    ;Params IlfProvider=kukaroboter.arctech.arconlin; Kuka.IsGlobalPoint=False; Kuka.PointName=P3; Kuka.BlendingEnabled=False; Kuka.MoveDataName=CPDAT1; Kuka.VelocityPath=0.5; Kuka.CurrentCDSetIndex=0; Kuka.MovementParameterFieldEnabled=True; ArcTech.WdatVarName=WDAT1; ArcTech.Basic=3.4.3.1264
  ;ENDFOLD
  $BWDSTART = FALSE
  LDAT_ACT = LCPDAT1
  FDAT_ACT = FP3
  BAS(#CP_PARAMS, 0.5)
  SET_CD_PARAMS (0)
  TRIGGER WHEN DISTANCE = 1 DELAY = ArcGetDelay(#PreDefinition, WDAT1) DO ArcMainNG(#PreDefinition, WDAT1, WP3) PRIO = -1
  TRIGGER WHEN PATH = ArcGetPath(#OnTheFlyArcOn, WDAT1) DELAY = ArcGetDelay(#GasPreflow, WDAT1) DO ArcMainNG(#GasPreflow, WDAT1, WP3) PRIO = -1
  TRIGGER WHEN PATH = ArcGetPath(#OnTheFlyArcOn, WDAT1) DELAY = 0 DO ArcMainNG(#ArcOnMoveStd, WDAT1, WP3) PRIO = -1
  ArcMainNG(#ArcOnBeforeMoveStd, WDAT1, WP3)
  LIN XP3
  ArcMainNG(#ArcOnAfterMoveStd, WDAT1, WP3)
;ENDFOLD
   $VEL.CP = 0.060
   LIN  {X -9.400, Y -9.400, Z 0.900, A 0.000, B 0.000, C 0.000} C_DIS
   $VEL.CP = 0.060
   LIN  {X 9.400, Y -9.400, Z 0.900, A 0.000, B 0.000, C 0.000} C_DIS
   $VEL.CP = 0.060
   LIN  {X 9.400, Y 9.400, Z 0.900, A 0.000, B 0.000, C 0.000} C_DIS
   $VEL.CP = 0.060
   LIN  {X -9.400, Y 9.400, Z 0.900, A 0.000, B 0.000, C 0.000} C_DIS

;FOLD ARCOFF WDAT2 LIN P4 CPDAT2 Tool[1]:cmttorch Base[1]:vrashatel ;%{PE}
  ;FOLD Parameters ;%{h}
    ;Params IlfProvider=kukaroboter.arctech.arcofflin; Kuka.IsGlobalPoint=False; Kuka.PointName=P4; Kuka.BlendingEnabled=False; Kuka.MoveDataName=CPDAT2; Kuka.VelocityPath=0.01; Kuka.CurrentCDSetIndex=0; Kuka.MovementParameterFieldEnabled=True; ArcTech.WdatVarName=WDAT2; ArcTech.Basic=3.4.3.1264
  ;ENDFOLD
  $BWDSTART = FALSE
  LDAT_ACT = LCPDAT2
  FDAT_ACT = FP4
  BAS(#CP_PARAMS, gArcBasVelDefinition)
  SET_CD_PARAMS (0)
  TRIGGER WHEN PATH = ArcGetPath(#ArcOffBefore, WDAT2) DELAY = 0 DO ArcMainNG(#ArcOffBeforeOffStd, WDAT2, WP4) PRIO = -1
  TRIGGER WHEN PATH = ArcGetPath(#OnTheFlyArcOff, WDAT2) DELAY = 0 DO ArcMainNG(#ArcOffMoveStd, WDAT2, WP4) PRIO = -1
  ArcMainNG(#ArcOffBeforeMoveStd, WDAT2, WP4)
  LIN XP4
  ArcMainNG(#ArcOffAfterMoveStd, WDAT2, WP4)
;ENDFOLD
   $VEL.CP = 0.080
   LIN  {X -9.040, Y 9.040, Z 0.900, A 0.000, B 0.000, C 0.000} C_DIS

;FOLD ARCON WDAT1 LIN P3 Vel=0.5 m/s CPDAT1 Tool[1]:cmttorch Base[1]:vrashatel ;%{PE}
  ;FOLD Parameters ;%{h}
    ;Params IlfProvider=kukaroboter.arctech.arconlin; Kuka.IsGlobalPoint=False; Kuka.PointName=P3; Kuka.BlendingEnabled=False; Kuka.MoveDataName=CPDAT1; Kuka.VelocityPath=0.5; Kuka.CurrentCDSetIndex=0; Kuka.MovementParameterFieldEnabled=True; ArcTech.WdatVarName=WDAT1; ArcTech.Basic=3.4.3.1264
  ;ENDFOLD
  $BWDSTART = FALSE
  LDAT_ACT = LCPDAT1
  FDAT_ACT = FP3
  BAS(#CP_PARAMS, 0.5)
  SET_CD_PARAMS (0)
  TRIGGER WHEN DISTANCE = 1 DELAY = ArcGetDelay(#PreDefinition, WDAT1) DO ArcMainNG(#PreDefinition, WDAT1, WP3) PRIO = -1
  TRIGGER WHEN PATH = ArcGetPath(#OnTheFlyArcOn, WDAT1) DELAY = ArcGetDelay(#GasPreflow, WDAT1) DO ArcMainNG(#GasPreflow, WDAT1, WP3) PRIO = -1
  TRIGGER WHEN PATH = ArcGetPath(#OnTheFlyArcOn, WDAT1) DELAY = 0 DO ArcMainNG(#ArcOnMoveStd, WDAT1, WP3) PRIO = -1
  ArcMainNG(#ArcOnBeforeMoveStd, WDAT1, WP3)
  LIN XP3
  ArcMainNG(#ArcOnAfterMoveStd, WDAT1, WP3)
;ENDFOLD
   $VEL.CP = 0.060
   LIN  {X -9.039, Y 5.102, Z 0.900, A 0.000, B 0.000, C 0.000} C_DIS
   $VEL.CP = 0.060
   LIN  {X -5.102, Y 9.039, Z 0.900, A 0.000, B 0.000, C 0.000} C_DIS
   $VEL.CP = 0.060
   LIN  {X -1.968, Y 9.039, Z 0.900, A 0.000, B 0.000, C 0.000} C_DIS
   $VEL.CP = 0.060
   LIN  {X 9.039, Y -1.968, Z 0.900, A 0.000, B 0.000, C 0.000} C_DIS
   $VEL.CP = 0.060
   LIN  {X 9.039, Y 1.968, Z 0.900, A 0.000, B 0.000, C 0.000} C_DIS
   $VEL.CP = 0.060
   LIN  {X -1.968, Y -9.039, Z 0.900, A 0.000, B 0.000, C 0.000} C_DIS
   $VEL.CP = 0.060
   LIN  {X -5.102, Y -9.039, Z 0.900, A 0.000, B 0.000, C 0.000} C_DIS
   $VEL.CP = 0.060
   LIN  {X -9.039, Y -5.102, Z 0.900, A 0.000, B 0.000, C 0.000} C_DIS
   $VEL.CP = 0.060
   LIN  {X -9.039, Y -9.039, Z 0.900, A 0.000, B 0.000, C 0.000} C_DIS
   $VEL.CP = 0.060
   LIN  {X 9.039, Y 9.039, Z 0.900, A 0.000, B 0.000, C 0.000} C_DIS
   $VEL.CP = 0.060
   LIN  {X 9.040, Y 9.040, Z 0.900, A 0.000, B 0.000, C 0.000} C_DIS
   $VEL.CP = 0.060
   LIN  {X 9.039, Y 5.102, Z 0.900, A 0.000, B 0.000, C 0.000} C_DIS
   $VEL.CP = 0.060
   LIN  {X 5.102, Y 9.039, Z 0.900, A 0.000, B 0.000, C 0.000} C_DIS
   $VEL.CP = 0.060
   LIN  {X 1.968, Y 9.039, Z 0.900, A 0.000, B 0.000, C 0.000} C_DIS
   $VEL.CP = 0.060
   LIN  {X -9.039, Y -1.968, Z 0.900, A 0.000, B 0.000, C 0.000} C_DIS
   $VEL.CP = 0.060
   LIN  {X -9.039, Y 1.968, Z 0.900, A 0.000, B 0.000, C 0.000} C_DIS
   $VEL.CP = 0.060
   LIN  {X 1.968, Y -9.039, Z 0.900, A 0.000, B 0.000, C 0.000} C_DIS
   $VEL.CP = 0.060
   LIN  {X 9.040, Y -9.040, Z 0.900, A 0.000, B 0.000, C 0.000} C_DIS

;FOLD ARCOFF WDAT2 LIN P4 CPDAT2 Tool[1]:cmttorch Base[1]:vrashatel ;%{PE}
  ;FOLD Parameters ;%{h}
    ;Params IlfProvider=kukaroboter.arctech.arcofflin; Kuka.IsGlobalPoint=False; Kuka.PointName=P4; Kuka.BlendingEnabled=False; Kuka.MoveDataName=CPDAT2; Kuka.VelocityPath=0.01; Kuka.CurrentCDSetIndex=0; Kuka.MovementParameterFieldEnabled=True; ArcTech.WdatVarName=WDAT2; ArcTech.Basic=3.4.3.1264
  ;ENDFOLD
  $BWDSTART = FALSE
  LDAT_ACT = LCPDAT2
  FDAT_ACT = FP4
  BAS(#CP_PARAMS, gArcBasVelDefinition)
  SET_CD_PARAMS (0)
  TRIGGER WHEN PATH = ArcGetPath(#ArcOffBefore, WDAT2) DELAY = 0 DO ArcMainNG(#ArcOffBeforeOffStd, WDAT2, WP4) PRIO = -1
  TRIGGER WHEN PATH = ArcGetPath(#OnTheFlyArcOff, WDAT2) DELAY = 0 DO ArcMainNG(#ArcOffMoveStd, WDAT2, WP4) PRIO = -1
  ArcMainNG(#ArcOffBeforeMoveStd, WDAT2, WP4)
  LIN XP4
  ArcMainNG(#ArcOffAfterMoveStd, WDAT2, WP4)
;ENDFOLD
   $VEL.CP = 0.080
   LIN  {X 9.039, Y -9.039, Z 0.900, A 0.000, B 0.000, C 0.000} C_DIS

